(* CODESYS project DBISFactory.project

Project tree, tasks and I/O mapping:
  Device : Berghof MX6 Control, Berghof Automation GmbH, version 1.16.2.0
    application Application
      libraries: Standard, * (System)
      task MainTask (cyclic, interval 4000 µs, priority 0) calls EtherCAT_Master.EtherCAT_Task [EtherCAT_Master.EtherCAT_Task], MAIN
      task EtherCAT_Master (cyclic, interval 4000 µs, priority 0) calls EtherCAT_Master.EtherCAT_Task [EtherCAT_Master.EtherCAT_Task]
      task VISU_TASK (cyclic, interval 100 ms, priority 31) calls VisuElems.Visu_Prg
      global variables SM
      program MAIN [SFC]: FU_Block_active, VG_Block_active, SL_Block_active, TC_active, HR_active, _aInit_active, INIT_BATCH_JOBS_active
      visualisation Visu
      HR/
        global variables HR
        program HR_MULTI_MODE [SFC]: STORE_BOX_active, GET_W_active, WAIT_FOR_VG_TO_PICK_UP_W_active, GET_BOX_active, DECIDE_active, STORE_W_active, WAIT_FOR_VG_TO_BRING_W_active, Init_active, TO_DEFAULT_POS_active
        FBs/
          function block HR_MOVE [ST]
          function block HR_STORE_W [ST]
          function block HR_MOVE_TO_POS [ST]
          function block HR_GET_W [ST]
          function block HR_PUT_W [ST]
          function block HR_TAKE_W [ST]
          function block HR_PUT_W_ON_CONVEYOR [ST]
          function block HR_TAKE_W_FROM_CONVEYOR [ST]
          function block HR_SWITCH_WS [ST]
        program HR_SINGLE_MODE [SFC]: HR_GET_W_active, ConveyorBack_HR_STORE_W_active_exit, HR_STORES_W_active, ConveyorBack_HR_STORE_W_active_active, HR_TO_DEFAULT_POS_active, HR_GET_W_entry, HR_TO_DEFAULT_POS_exit, HR_GETS_W_exit, HR_CONVEYOR_BACKWARD_active, Store_W_active, ToDefaultPos_HR_STORE_W_active_active, HR_WAIT_FOR_TC_active, HR_CONVEYOR_BACKWARD_exit, Init_active, ConveyorBack_HR_STORE_W_active_entry, HR_CALIBRATE_Y_AXIS_active, HR_CALIBRATE_Y_AXIS_exit, HR_CONVEYOR_FORWARD_exit, HR_CONVEYOR_FORWARD_active, HR_STORES_W_exit, HR_SET_TC_STATE_exit, HR_SET_TC_STATE_active
        program HR_SORTING_MODE [SFC]: SORTING_active, TO_DEFAULT_POS_exit, TO_DEFAULT_POS_active, Init_active, HR_SET_TC_STATE_active, HR_SET_TC_STATE_exit, TO_DEFAULT_POS_2_exit, TO_DEFAULT_POS_2_active
      VG/
        FBs/
          function block VG_MOVE [ST]
          function block VG_MOVE_TO_POS [ST]
        program VG_MULTI_MODE [SFC]: TO_DEFAULT_POS_active, DECIDE_active, FROM_HR_TO_FUR_active, TO_SL_TAKE_W_active, TO_HR_PUT_W_active, TO_HR_TAKE_W_active, TO_EJECT_active, Init_active
        program VG_SINGLE_MODE [SFC]: XForward_VG_TAKE_W_active_exit, YUp_VG_DROP_W_active_exit, VG_TO_FU_entry, ZBack_VG_FROM_SL_TO_HR_active_exit, Suction_VG_TAKE_W_active_active, ZBack_VG_TO_FU_active_active, VG_TO_SL_active, YDown_VG_TO_FU_active_exit, ZBack_VG_TO_FU_active_exit_0, Wait_VG_DROP_W_active_active, XForward_VG_TAKE_W_active_active, Wait_VG_TO_FU_active_exit, YDown_VG_DROP_W_active_active, VG_TO_EJECT_POINT_active, YDown_VG_DROP_W_active_exit, OpenVentil_VG_DROP_W_active_exit, VG_EJECT_W_active, OpenVentil_VG_DROP_W_active_active, ZBack_VG_FROM_SL_TO_HR_active_active, ZLeft_AND_XForward_VG_TO_FU_active_active, YDown_VG_TAKE_W_active_exit, YUp_VG_TO_FU_active_exit, YUp_VG_TAKE_W_active_exit, Init_active, YDown_VG_TO_FU_active_active, ZBack_VG_TO_FU_active_exit, YUp_VG_TO_FU_active_active, ZBack_VG_TAKE_W_active_exit, VG_TO_FU_active, OpenVentil_VG_TO_FU_active_active, YUp_VG_DROP_W_active_active, ZBack_VG_TAKE_W_active_active, VG_TAKE_W_entry, Wait_VG_TO_FU_active_active, YUp_VG_TAKE_W_active_active, VG_DROP_W_entry, VG_TO_DEFAULT_POS_active, VG_DROP_W_active, VG_TAKE_W_active, YDown_VG_TAKE_W_active_active, Wait_VG_DROP_W_active_exit, VG_DROP_W_exit, VG_FROM_SL_TO_HR_active, VG_TO_HR_active, ZBack_VG_TO_FU_active_active_0, ZLeft_AND_XForward_VG_TO_FU_active_exit, VG_WAIT_FOR_SL_active, VG_WAIT_FOR_SL_exit, VG_YUp_active, VG_YUp_exit, VG_TO_EJECT_POINT_exit, VG_EJECT_active, VG_EJECT_exit, BACK_TO_DEFAULT_active, VG_TO_SL_exit, VG_DIRECTLY_EJECT_W_active, VG_TO_HR_exit
        global variables VG
      FUR/
        program FUR_SINGLE_MODE [SFC]: FUR_SUCCER_UP_active_0, FUR_SUCCER_TO_ROTATION_DESK_active, FUR_SAW_active, FUR_WAIT_FOR_W_exit, Init_active, FUR_SUCCER_DOWN2_active, FUR_SUCCER_DOWN_active, FUR_TO_CONVEYOR_active, FUR_SUCCER_UP_active, FUR_TO_DEFAULT_POS_active, FUR_WAIT_FOR_W_active, FUR_BURN_active
        program FUR_MULTI_MODE [SFC]: BURNER_active, SUCCER_active, SAW_active, TO_DEFAULT_POS_active, TO_DEFAULT_POS_exit
        global variables FUR
        FBs/
          function block FUR_BURN [ST]
      SL/
        program SL_SINGLE_MODE [SFC]: Init_active, SL_GO_active
        global variables SL
        program SL_MULTI_MODE [SFC]: SL_GO_active, Init_active
        FBs/
          function block SL_FB [SFC]: Init_active, SL_COLORCHECK_active, SL_GET_VALUE_active, SL_PASS_LBEntry_active, SL_PASS_LBEntry_exit, SL_PULS_COUNTER_active, SL_PULS_COUNTER_exit, SL_SORTING_active, SL_STOREROOM_active
      TC/
        FUNs/
          function addBatchJobToQueue [ST]
          function newWorkpiece [ST]
          function addWorkpieceToBatchJob [ST]
          function newFormat [ST]
          function newBatchJob [ST]
        global variables TC
        program TC_POU [SFC]: Decide_next_W_or_BatchJob_active, Set_Workpiece_active, start_batch_job_active, Init_active, Next_W_active, Next_W_exit, Decide_next_W_or_BatchJob_exit, Start_Batch_Job_exit
      datastructures/
        Enums/
          data type ExecutionMode
          data type RackPos
          States/
            data type BatchJobState
            data type HR_State
            data type VG_State
            data type FUR_State
            data type SL_State
            data type W_State
            data type TC_State
        Structs/
          data type Format
          data type BatchJobQueue
          data type Workpiece
          data type BatchJob
      Symbols
    Extension_Slots : Extension Slots, Berghof Automation GmbH, order no. 
      , version 1.0.0.0
      <Leer>
      Berghof_IO : Berghof IO, Berghof Automation GmbH, order no. 
      , version 1.1.0.0
          unmapped channels: Digital Input 0, Digital Input 1, Digital Input 2, Digital Input 3, Digital Input 4, Digital Output 0, Digital Output 1, Digital Output 2, Digital Output 3, Digital Output 4, Channel 0, Channel 1, Channel 2, Channel 3, Channel 4, Channel 5, Channel 6, Channel 7, Channel 8, Channel 9, Channel 10, Channel 11, Channel 0, Channel 1, Channel 2, Channel 3, Channel 4, Channel 5, Channel 6, Channel 7, Counter/Encoder 0, Counter/Encoder 1, Counter/Encoder 2, DUMMY 0
    EtherCAT_Master : EtherCAT Master, 3S - Smart Software Solutions GmbH, version 3.5.10.0
        settings: SlaveAutoRestart = True; NetworkName = 'eth1'; SelectNetworkByName = True
      ECC_DIO_16_16P : ECC DIO 16/16 P (250 000 600), Berghof Automation GmbH, version Revision=16#00000001
          settings: DC sync0 cycletime = 4000; DC sync1 cycletime = 4000
          unmapped channels: Digital Output 0, Digital Output 1, Digital Input 0, Digital Input 1
  libraries: VisuSymbols, 3.5.10.0 (System)
  text list GlobalTextList
*)

// Device/Application/datastructures/Enums/States/BatchJobState
(*
	States of a BatchJob

Copyright (c) 2019 Manuel Goester, Michael Witt, Klaus Kammerer
Institute of Databases and Information Systems, Ulm University, Germany

Permission is hereby granted, free of charge, to any person obtaining a copy 
of this software and associated documentation files (the "Software"), to deal 
in the Software without restriction, including without limitation the rights 
to use, copy, modify, merge, publish, distribute, sublicense, and/or sell 
copies of the Software, and to permit persons to whom the Software is 
furnished to do so, subject to the following conditions:

The above copyright notice and this permission notice shall be included in 
all copies or substantial portions of the Software.

THE SOFTWARE IS PROVIDED "AS IS", WITHOUT WARRANTY OF ANY KIND, EXPRESS OR 
IMPLIED, INCLUDING BUT NOT LIMITED TO THE WARRANTIES OF MERCHANTABILITY, 
FITNESS FOR A PARTICULAR PURPOSE AND NONINFRINGEMENT. IN NO EVENT SHALL THE 
AUTHORS OR COPYRIGHT HOLDERS BE LIABLE FOR ANY CLAIM, DAMAGES OR OTHER 
LIABILITY, WHETHER IN AN ACTION OF CONTRACT, TORT OR OTHERWISE, ARISING FROM, 
OUT OF OR IN CONNECTION WITH THE SOFTWARE OR THE USE OR OTHER DEALINGS 
IN THE SOFTWARE.
*)
TYPE BatchJobState :
(
	// NULL always expresses that the object has not been initialized yet
	NULL := 0,
	
	// BatchJob has been initialized and is waiting to be executed
	WAITING := 1,
	
	// BatchJob has been started and is being executed now
	STARTED := 2,
	
	// BatchJob has been paused during execution
	PAUSED := 3,
	
	// BatchJob has been aborted. This may happen at any time
	ABORTED := 4,
	
	// BatchJob has been finished
	FINISHED := 5
);
END_TYPE

// Device/Application/datastructures/Enums/ExecutionMode
(*
	Execution modes of a BatchJob
	
Copyright (c) 2019 Manuel Goester, Michael Witt, Klaus Kammerer
Institute of Databases and Information Systems, Ulm University, Germany

Permission is hereby granted, free of charge, to any person obtaining a copy 
of this software and associated documentation files (the "Software"), to deal 
in the Software without restriction, including without limitation the rights 
to use, copy, modify, merge, publish, distribute, sublicense, and/or sell 
copies of the Software, and to permit persons to whom the Software is 
furnished to do so, subject to the following conditions:

The above copyright notice and this permission notice shall be included in 
all copies or substantial portions of the Software.

THE SOFTWARE IS PROVIDED "AS IS", WITHOUT WARRANTY OF ANY KIND, EXPRESS OR 
IMPLIED, INCLUDING BUT NOT LIMITED TO THE WARRANTIES OF MERCHANTABILITY, 
FITNESS FOR A PARTICULAR PURPOSE AND NONINFRINGEMENT. IN NO EVENT SHALL THE 
AUTHORS OR COPYRIGHT HOLDERS BE LIABLE FOR ANY CLAIM, DAMAGES OR OTHER 
LIABILITY, WHETHER IN AN ACTION OF CONTRACT, TORT OR OTHERWISE, ARISING FROM, 
OUT OF OR IN CONNECTION WITH THE SOFTWARE OR THE USE OR OTHER DEALINGS 
IN THE SOFTWARE.
*)
TYPE ExecutionMode :
(
	single := 0,
	multi := 1,
	sorting := 2
);
END_TYPE

// Device/Application/datastructures/Structs/Format
(*
	A Format defines the execution options of a workpiece

Copyright (c) 2019 Manuel Goester, Michael Witt, Klaus Kammerer
Institute of Databases and Information Systems, Ulm University, Germany

Permission is hereby granted, free of charge, to any person obtaining a copy 
of this software and associated documentation files (the "Software"), to deal 
in the Software without restriction, including without limitation the rights 
to use, copy, modify, merge, publish, distribute, sublicense, and/or sell 
copies of the Software, and to permit persons to whom the Software is 
furnished to do so, subject to the following conditions:

The above copyright notice and this permission notice shall be included in 
all copies or substantial portions of the Software.

THE SOFTWARE IS PROVIDED "AS IS", WITHOUT WARRANTY OF ANY KIND, EXPRESS OR 
IMPLIED, INCLUDING BUT NOT LIMITED TO THE WARRANTIES OF MERCHANTABILITY, 
FITNESS FOR A PARTICULAR PURPOSE AND NONINFRINGEMENT. IN NO EVENT SHALL THE 
AUTHORS OR COPYRIGHT HOLDERS BE LIABLE FOR ANY CLAIM, DAMAGES OR OTHER 
LIABILITY, WHETHER IN AN ACTION OF CONTRACT, TORT OR OTHERWISE, ARISING FROM, 
OUT OF OR IN CONNECTION WITH THE SOFTWARE OR THE USE OR OTHER DEALINGS 
IN THE SOFTWARE.
*)
TYPE Format :
STRUCT
	furEnabled: BOOL;
	sawEnabled: BOOL;
	colorCheckEnabled: BOOL;
	ejectEnabled: BOOL;
	
	furDuration: TIME;
	sawDuration: TIME;
END_STRUCT
END_TYPE

// Device/Application/datastructures/Structs/BatchJobQueue
(*
	Configured BatchJobs are stored in a BatchJobQueue

Copyright (c) 2019 Manuel Goester, Michael Witt, Klaus Kammerer
Institute of Databases and Information Systems, Ulm University, Germany

Permission is hereby granted, free of charge, to any person obtaining a copy 
of this software and associated documentation files (the "Software"), to deal 
in the Software without restriction, including without limitation the rights 
to use, copy, modify, merge, publish, distribute, sublicense, and/or sell 
copies of the Software, and to permit persons to whom the Software is 
furnished to do so, subject to the following conditions:

The above copyright notice and this permission notice shall be included in 
all copies or substantial portions of the Software.

THE SOFTWARE IS PROVIDED "AS IS", WITHOUT WARRANTY OF ANY KIND, EXPRESS OR 
IMPLIED, INCLUDING BUT NOT LIMITED TO THE WARRANTIES OF MERCHANTABILITY, 
FITNESS FOR A PARTICULAR PURPOSE AND NONINFRINGEMENT. IN NO EVENT SHALL THE 
AUTHORS OR COPYRIGHT HOLDERS BE LIABLE FOR ANY CLAIM, DAMAGES OR OTHER 
LIABILITY, WHETHER IN AN ACTION OF CONTRACT, TORT OR OTHERWISE, ARISING FROM, 
OUT OF OR IN CONNECTION WITH THE SOFTWARE OR THE USE OR OTHER DEALINGS 
IN THE SOFTWARE.
*)
TYPE BatchJobQueue :
STRUCT
	// batch job queue
	batchJobs: ARRAY [1..512] OF BatchJob;
	
	// next free place in batchJobs
	nextFreePos: INT := 1;
	
	// amount of batch jobs currently being in queue
	amountBatchJobs: INT := 0;
	
	// true if batchJobs array full
	full: BOOL;
END_STRUCT
END_TYPE

// Device/Application/datastructures/Structs/Workpiece
(*
	Datastructure describing the "real world workpiece"

Copyright (c) 2019 Manuel Goester, Michael Witt, Klaus Kammerer
Institute of Databases and Information Systems, Ulm University, Germany

Permission is hereby granted, free of charge, to any person obtaining a copy 
of this software and associated documentation files (the "Software"), to deal 
in the Software without restriction, including without limitation the rights 
to use, copy, modify, merge, publish, distribute, sublicense, and/or sell 
copies of the Software, and to permit persons to whom the Software is 
furnished to do so, subject to the following conditions:

The above copyright notice and this permission notice shall be included in 
all copies or substantial portions of the Software.

THE SOFTWARE IS PROVIDED "AS IS", WITHOUT WARRANTY OF ANY KIND, EXPRESS OR 
IMPLIED, INCLUDING BUT NOT LIMITED TO THE WARRANTIES OF MERCHANTABILITY, 
FITNESS FOR A PARTICULAR PURPOSE AND NONINFRINGEMENT. IN NO EVENT SHALL THE 
AUTHORS OR COPYRIGHT HOLDERS BE LIABLE FOR ANY CLAIM, DAMAGES OR OTHER 
LIABILITY, WHETHER IN AN ACTION OF CONTRACT, TORT OR OTHERWISE, ARISING FROM, 
OUT OF OR IN CONNECTION WITH THE SOFTWARE OR THE USE OR OTHER DEALINGS 
IN THE SOFTWARE.
*)
TYPE Workpiece :
STRUCT
	// red, blue, white or unknown
	color: STRING[7];
	
	// 0 = high rack, 1 = vacuum gripper, 2 = Furnace, 3 = sorting line
	linePos: INT;
	
	// position in high rack at begin and end of batch job
	// (1,1) (1,2) (1,3)
	// (2,1) (2,2) (2,3)
	// (3,1) (3,2) (3,3)
	//highRackPos: ARRAY [1..2] OF INT;
	//highRackPosEnd: ARRAY [1..2] OF INT;
	
	// position in sorting line
	sortingLinePos: INT;
	
	state: W_State;	
	startPos: RackPos;
	endPos: RackPos;
	
	// defines which actions will be executed and how long
	format: Format;
END_STRUCT
END_TYPE

// Device/Application/datastructures/Structs/BatchJob
(*
	A BatchJob is a task which shall be executed on the production lane. 
	It consists of a set of workpieces, which are executed by the production lane in a certain mode.

Copyright (c) 2019 Manuel Goester, Michael Witt, Klaus Kammerer
Institute of Databases and Information Systems, Ulm University, Germany

Permission is hereby granted, free of charge, to any person obtaining a copy 
of this software and associated documentation files (the "Software"), to deal 
in the Software without restriction, including without limitation the rights 
to use, copy, modify, merge, publish, distribute, sublicense, and/or sell 
copies of the Software, and to permit persons to whom the Software is 
furnished to do so, subject to the following conditions:

The above copyright notice and this permission notice shall be included in 
all copies or substantial portions of the Software.

THE SOFTWARE IS PROVIDED "AS IS", WITHOUT WARRANTY OF ANY KIND, EXPRESS OR 
IMPLIED, INCLUDING BUT NOT LIMITED TO THE WARRANTIES OF MERCHANTABILITY, 
FITNESS FOR A PARTICULAR PURPOSE AND NONINFRINGEMENT. IN NO EVENT SHALL THE 
AUTHORS OR COPYRIGHT HOLDERS BE LIABLE FOR ANY CLAIM, DAMAGES OR OTHER 
LIABILITY, WHETHER IN AN ACTION OF CONTRACT, TORT OR OTHERWISE, ARISING FROM, 
OUT OF OR IN CONNECTION WITH THE SOFTWARE OR THE USE OR OTHER DEALINGS 
IN THE SOFTWARE.
*)
TYPE BatchJob :
STRUCT
	// amount of workpieces in batch job
	batchSize: INT;
	
	// workpieces being processed
	workpieces: ARRAY [1..9] OF Workpiece;
	
	// next free place in workpieces
	nextFreeWPos: INT := 1;
	
	// index in workpieces of the next workpiece whose production has not started yet
	nextNotProcessedIdx: INT := 1;
	
	// states how many workpieces are already finished
	amountFinishedW: INT := 0;
	
	// type of execution
	mode: ExecutionMode := ExecutionMode.single;
	
	// time when created
	timeCreated: DATE_AND_TIME;
	
	// time when started
	timeStarted: DATE_AND_TIME;
	
	// time when finished / aborted
	timeFinished: DATE_AND_TIME;
	
	// states the time how long the batch job was in pause state
	pauseDuration: TIME;
	
	// states how long the batch job took 
	duration: TIME;
	
	// state of batch job
	state: BatchJobState := BatchJobState.NULL;
END_STRUCT
END_TYPE

// Device/Application/datastructures/Enums/RackPos
(*
	Positions in high rack. Used for HR navigation

Copyright (c) 2019 Manuel Goester, Michael Witt, Klaus Kammerer
Institute of Databases and Information Systems, Ulm University, Germany

Permission is hereby granted, free of charge, to any person obtaining a copy 
of this software and associated documentation files (the "Software"), to deal 
in the Software without restriction, including without limitation the rights 
to use, copy, modify, merge, publish, distribute, sublicense, and/or sell 
copies of the Software, and to permit persons to whom the Software is 
furnished to do so, subject to the following conditions:

The above copyright notice and this permission notice shall be included in 
all copies or substantial portions of the Software.

THE SOFTWARE IS PROVIDED "AS IS", WITHOUT WARRANTY OF ANY KIND, EXPRESS OR 
IMPLIED, INCLUDING BUT NOT LIMITED TO THE WARRANTIES OF MERCHANTABILITY, 
FITNESS FOR A PARTICULAR PURPOSE AND NONINFRINGEMENT. IN NO EVENT SHALL THE 
AUTHORS OR COPYRIGHT HOLDERS BE LIABLE FOR ANY CLAIM, DAMAGES OR OTHER 
LIABILITY, WHETHER IN AN ACTION OF CONTRACT, TORT OR OTHERWISE, ARISING FROM, 
OUT OF OR IN CONNECTION WITH THE SOFTWARE OR THE USE OR OTHER DEALINGS 
IN THE SOFTWARE.
*)
TYPE RackPos :
(
	NULL := 0,
	RACK_11 := 1,
	RACK_12 := 2,
	RACK_13 := 3,
	RACK_21 := 4,
	RACK_22 := 5,
	RACK_23 := 6,
	RACK_31 := 7,
	RACK_32 := 8,
	RACK_33 := 9,
	
	CONVEYOR := 10,
	
	// there are different values for up position or down position at rack or at conveyor
	// see: HR_FBs/HR_MOVE_TO_POS
	UP := 11,
	DOWN := 12	
);
END_TYPE

// Device/Application/datastructures/Enums/States/HR_State
(*
	States of the HR (High Rack) station.

Copyright (c) 2019 Manuel Goester, Michael Witt, Klaus Kammerer
Institute of Databases and Information Systems, Ulm University, Germany

Permission is hereby granted, free of charge, to any person obtaining a copy 
of this software and associated documentation files (the "Software"), to deal 
in the Software without restriction, including without limitation the rights 
to use, copy, modify, merge, publish, distribute, sublicense, and/or sell 
copies of the Software, and to permit persons to whom the Software is 
furnished to do so, subject to the following conditions:

The above copyright notice and this permission notice shall be included in 
all copies or substantial portions of the Software.

THE SOFTWARE IS PROVIDED "AS IS", WITHOUT WARRANTY OF ANY KIND, EXPRESS OR 
IMPLIED, INCLUDING BUT NOT LIMITED TO THE WARRANTIES OF MERCHANTABILITY, 
FITNESS FOR A PARTICULAR PURPOSE AND NONINFRINGEMENT. IN NO EVENT SHALL THE 
AUTHORS OR COPYRIGHT HOLDERS BE LIABLE FOR ANY CLAIM, DAMAGES OR OTHER 
LIABILITY, WHETHER IN AN ACTION OF CONTRACT, TORT OR OTHERWISE, ARISING FROM, 
OUT OF OR IN CONNECTION WITH THE SOFTWARE OR THE USE OR OTHER DEALINGS 
IN THE SOFTWARE.
*)
TYPE HR_State :
(
	// NULL always expresses that the Object has not been initialized yet
	NULL := 0,
	
	// used in single mode
	AT_DEFAULT_POS := 1,
	FINISHED_SINGLE_MODE := 2,
	AT_CONVEYOR_BOX_FULL := 25,
	AT_CONVEYOR_BOX_EMPTY := 26,
	
	// used in multi mode
	WAIT_FOR_VG_TO_BRING_W := 8,
	GET_W := 9, // <-- also used in single mode
	GET_BOX := 10,
	STORE_W := 20,
	STORE_BOX := 19,
	WAIT_FOR_VG_TO_PICK_UP_W := 11,
	READY := 12,
	
	// used in sorting mode
	FINISHED_SORTING_MODE := 40,
	SORTING := 41
);
END_TYPE

// Device/Application/datastructures/Enums/States/VG_State
(*
	States of the VG (Vacuum Gripper) station.

Copyright (c) 2019 Manuel Goester, Michael Witt, Klaus Kammerer
Institute of Databases and Information Systems, Ulm University, Germany

Permission is hereby granted, free of charge, to any person obtaining a copy 
of this software and associated documentation files (the "Software"), to deal 
in the Software without restriction, including without limitation the rights 
to use, copy, modify, merge, publish, distribute, sublicense, and/or sell 
copies of the Software, and to permit persons to whom the Software is 
furnished to do so, subject to the following conditions:

The above copyright notice and this permission notice shall be included in 
all copies or substantial portions of the Software.

THE SOFTWARE IS PROVIDED "AS IS", WITHOUT WARRANTY OF ANY KIND, EXPRESS OR 
IMPLIED, INCLUDING BUT NOT LIMITED TO THE WARRANTIES OF MERCHANTABILITY, 
FITNESS FOR A PARTICULAR PURPOSE AND NONINFRINGEMENT. IN NO EVENT SHALL THE 
AUTHORS OR COPYRIGHT HOLDERS BE LIABLE FOR ANY CLAIM, DAMAGES OR OTHER 
LIABILITY, WHETHER IN AN ACTION OF CONTRACT, TORT OR OTHERWISE, ARISING FROM, 
OUT OF OR IN CONNECTION WITH THE SOFTWARE OR THE USE OR OTHER DEALINGS 
IN THE SOFTWARE.
*)
TYPE VG_State :
(
	// NULL always expresses that the object has not been initialized yet
	NULL := 0,
	
	// used in single mode
	FROM_HR_TO_EJECT := 6,
	AT_HR := 30,
	FROM_HR_TO_FUR := 31,
	AT_SL_OUTPUT_1 := 32,
	AT_SL_OUTPUT_2 := 33,
	AT_SL_OUTPUT_3 := 34,
	WAIT_FOR_SL := 35,
	AT_EJECT_1 := 36,
	AT_EJECT_2 := 37,
	AT_EJECT_3 := 38,
	TO_SL_OUTPUT_1 := 39,
	TO_SL_OUTPUT_2 := 40,
	TO_SL_OUTPUT_3 := 41,
	FROM_DEFAULT_POS_TO_HR := 43,
	GET_W_FROM_HR := 44,
	ABOVE_SL := 56,
	FROM_SL_TO_HR := 57,
	DROPPING_W_TO_HR := 59,
	
	// used in multi mode
	TO_FUR_PUT_W := 8,
	TO_FUR_PUT_W_FINISHED := 9,
	TO_SL_TAKE_W := 10,
	TO_SL_TAKE_W_FINISHED := 11,
	TO_HR_PUT_W := 12,
	TO_HR_PUT_W_FINISHED := 13,
	TO_HR_TAKE_W := 14,
	TO_HR_TAKE_W_FINISHED := 15,
	TO_EJECT := 16,
	TO_EJECT_FINISHED := 17,
	TO_SL := 45,
	// ready if VG is at default pos or if VG put down a workpiece at HR --> VG is ready for next workpiece
	READY := 18,
	
	// used in single and multi mode
	AT_DEFAULT_POS := 1,
	TO_DEFAULT_POS := 5
);
END_TYPE

// Device/Application/datastructures/Enums/States/FUR_State
(*
	States of the FUR (Furnace) station.
	The station is composed of a burner, succer, rotary desk and saw.

Copyright (c) 2019 Manuel Goester, Michael Witt, Klaus Kammerer
Institute of Databases and Information Systems, Ulm University, Germany

Permission is hereby granted, free of charge, to any person obtaining a copy 
of this software and associated documentation files (the "Software"), to deal 
in the Software without restriction, including without limitation the rights 
to use, copy, modify, merge, publish, distribute, sublicense, and/or sell 
copies of the Software, and to permit persons to whom the Software is 
furnished to do so, subject to the following conditions:

The above copyright notice and this permission notice shall be included in 
all copies or substantial portions of the Software.

THE SOFTWARE IS PROVIDED "AS IS", WITHOUT WARRANTY OF ANY KIND, EXPRESS OR 
IMPLIED, INCLUDING BUT NOT LIMITED TO THE WARRANTIES OF MERCHANTABILITY, 
FITNESS FOR A PARTICULAR PURPOSE AND NONINFRINGEMENT. IN NO EVENT SHALL THE 
AUTHORS OR COPYRIGHT HOLDERS BE LIABLE FOR ANY CLAIM, DAMAGES OR OTHER 
LIABILITY, WHETHER IN AN ACTION OF CONTRACT, TORT OR OTHERWISE, ARISING FROM, 
OUT OF OR IN CONNECTION WITH THE SOFTWARE OR THE USE OR OTHER DEALINGS 
IN THE SOFTWARE.
*)
TYPE FUR_State :
(
	// TODO : Use these states also in multi mode
	
	// NULL always expresses that the Object has not been initialized yet
	NULL := 0,
	
	// used in single mode
	// FUR is ready to take a new workpiece
	FUR_WAITING_FOR_W := 1,	
	// Workpiece passed the lightbarrier at waggon
	FUR_LB_PASSED := 2,
	
	// used in single and multi mode
	// Wagon is inside of burner
	FUR_WAGON_INSIDE := 3,
	// Furnace is finished with buring the workpiece
	FUR_BURNED := 4,
	// Wagon is outside of burner
	FUR_WAGON_OUTSIDE := 5,	
	
	// used in single mode
	// furnace succer is at furnace
	FUR_SUCCER_AT_FUR := 6,
	// furnace succer picks up workpiece
	FUR_SUCCER_DOWN_AT_FUR := 7,
	FUR_SUCCER_UP_AT_FUR := 8,
	// furnace succer on the way to rotary desk
	FUR_SUCCER_TO_ROTARY_DESK := 9,
	// furnace succer at rotary desk
	FUR_SUCCER_AT_ROTARY_DESK := 10,
	// furnace succer puts down workpiece
	FUR_SUCCER_DOWN_AT_RD := 11,
	FUR_SUCCER_UP_AT_RD := 12,
	// saw has been finished
	FUR_SAW_FINISHED := 13,	
	// saw has been skipped			
	FUR_SKIP_SAW := 14,
	// station has finished processing this workpiece
	FUR_W_FINISHED_BACK_TO_DEFAULT := 15
);
END_TYPE

// Device/Application/datastructures/Enums/States/SL_State
(*
	States of the SL (Sorting Line) station.

Copyright (c) 2019 Manuel Goester, Michael Witt, Klaus Kammerer
Institute of Databases and Information Systems, Ulm University, Germany

Permission is hereby granted, free of charge, to any person obtaining a copy 
of this software and associated documentation files (the "Software"), to deal 
in the Software without restriction, including without limitation the rights 
to use, copy, modify, merge, publish, distribute, sublicense, and/or sell 
copies of the Software, and to permit persons to whom the Software is 
furnished to do so, subject to the following conditions:

The above copyright notice and this permission notice shall be included in 
all copies or substantial portions of the Software.

THE SOFTWARE IS PROVIDED "AS IS", WITHOUT WARRANTY OF ANY KIND, EXPRESS OR 
IMPLIED, INCLUDING BUT NOT LIMITED TO THE WARRANTIES OF MERCHANTABILITY, 
FITNESS FOR A PARTICULAR PURPOSE AND NONINFRINGEMENT. IN NO EVENT SHALL THE 
AUTHORS OR COPYRIGHT HOLDERS BE LIABLE FOR ANY CLAIM, DAMAGES OR OTHER 
LIABILITY, WHETHER IN AN ACTION OF CONTRACT, TORT OR OTHERWISE, ARISING FROM, 
OUT OF OR IN CONNECTION WITH THE SOFTWARE OR THE USE OR OTHER DEALINGS 
IN THE SOFTWARE.
*)
TYPE SL_State :
(
	
	// NULL always expresses that the object has not been initialized yet
	NULL := 0,
	
	// SL is ready to process a new workpiece
	WAITING_FOR_W := 1,
	// Lightbarrier at SL entry has been passed by a workpiece
	W_AT_LB := 2,

	W_AT_COLORCHECK := 3,
	COLORCHECK_FINISHED := 4,
	W_READY_FOR_SORTING := 5,
	// if no color was detected, the workpiece will be thrown out to trash 
	THROW_OUT := 6,
	
	SORTING := 7,
	WAITING_FOR_VG_TO_PICK_UP_W	 := 8,
	EJECT := 9,
	EJECTED := 10,
	
	// SL got a workpiece to process it
	W_RECEIVED := 11
);
END_TYPE

// Device/Application/datastructures/Enums/States/W_State
(*
	Workpiece States

Copyright (c) 2019 Manuel Goester, Michael Witt, Klaus Kammerer
Institute of Databases and Information Systems, Ulm University, Germany

Permission is hereby granted, free of charge, to any person obtaining a copy 
of this software and associated documentation files (the "Software"), to deal 
in the Software without restriction, including without limitation the rights 
to use, copy, modify, merge, publish, distribute, sublicense, and/or sell 
copies of the Software, and to permit persons to whom the Software is 
furnished to do so, subject to the following conditions:

The above copyright notice and this permission notice shall be included in 
all copies or substantial portions of the Software.

THE SOFTWARE IS PROVIDED "AS IS", WITHOUT WARRANTY OF ANY KIND, EXPRESS OR 
IMPLIED, INCLUDING BUT NOT LIMITED TO THE WARRANTIES OF MERCHANTABILITY, 
FITNESS FOR A PARTICULAR PURPOSE AND NONINFRINGEMENT. IN NO EVENT SHALL THE 
AUTHORS OR COPYRIGHT HOLDERS BE LIABLE FOR ANY CLAIM, DAMAGES OR OTHER 
LIABILITY, WHETHER IN AN ACTION OF CONTRACT, TORT OR OTHERWISE, ARISING FROM, 
OUT OF OR IN CONNECTION WITH THE SOFTWARE OR THE USE OR OTHER DEALINGS 
IN THE SOFTWARE.
*)
TYPE W_State :
(
	// NULL always expresses that the object has not been initialized yet
	NULL := 0,
	
	// states at HR
	AT_RACK_11 := 111,
	AT_RACK_12 := 112,
	AT_RACK_13 := 113,
	AT_RACK_21 := 121,
	AT_RACK_22 := 122,
	AT_RACK_23 := 123,
	AT_RACK_31 := 131,
	AT_RACK_32 := 132,
	AT_RACK_33 := 133,
	
	// NOT used
	FROM_RACK_TO_CONVEYOR := 140,
	AT_CONVEYOR_INSIDE := 141,
	FROM_CONVEYOR_INSIDE_TO_OUTSIDE := 142,
	AT_CONVEYOR_OUTSIDE := 143,
	FROM_CONVEYOR_OUTSIDE_TO_INSIDE := 144,
	
	// states at VG
	// NOT used
	AT_HR := 200,
	FROM_HR_TO_FUR := 201,
	FROM_SL_OUTPUT_TO_HR := 202,
	FROM_SL_OUTPUT_1_TO_HR := 203,
	FROM_SL_OUTPUT_2_TO_HR := 204,
	FROM_SL_OUTPUT_3_TO_HR := 205,
	FROM_SL_TO_EJECT := 206,
	FROM_SL_OUTPUT_1_TO_EJECT := 207,
	FROM_SL_OUTPUT_2_TO_EJECT := 208,
	FROM_SL_OUTPUT_3_TO_EJECT := 209,
	FROM_FUR_TO_HR := 210,
	
	// states at FUR
	AT_FUR_IN_WAGON := 300,
	AT_FUR_IN_FUR := 301,
	AT_FUR_ATTACHED_TO_SUCCER := 302,
	AT_FUR_ON_ROTARY_DESK := 303,
	AT_FUR_AT_SAW := 304,
	AT_FUR_ON_CONVEYOR := 305,
	
	// states at SL
	// not used
	AT_SL_AT_ENTRY_LIGHT_BARRIER := 400,
	AT_SL_AT_COLORCHECK := 401,
	AT_SL_AT_EXIT_LIGHT_BARRIER := 402,
	AT_SL_OUTPUT_1 := 403,
	AT_SL_OUTPUT_2 := 404,
	AT_SL_OUTPUT_3 := 405,
	AT_SL_OUTPUT_TRASH := 406,
	
	// states at EJECT point
	// not used
	AT_EJECT_1 := 500,
	AT_EJECT_2 := 501,
	AT_EJECT_3 := 502
);
END_TYPE

// Device/Application/datastructures/Enums/States/TC_State
(*
	States of TC (Task Configurator).

Copyright (c) 2019 Manuel Goester, Michael Witt, Klaus Kammerer
Institute of Databases and Information Systems, Ulm University, Germany

Permission is hereby granted, free of charge, to any person obtaining a copy 
of this software and associated documentation files (the "Software"), to deal 
in the Software without restriction, including without limitation the rights 
to use, copy, modify, merge, publish, distribute, sublicense, and/or sell 
copies of the Software, and to permit persons to whom the Software is 
furnished to do so, subject to the following conditions:

The above copyright notice and this permission notice shall be included in 
all copies or substantial portions of the Software.

THE SOFTWARE IS PROVIDED "AS IS", WITHOUT WARRANTY OF ANY KIND, EXPRESS OR 
IMPLIED, INCLUDING BUT NOT LIMITED TO THE WARRANTIES OF MERCHANTABILITY, 
FITNESS FOR A PARTICULAR PURPOSE AND NONINFRINGEMENT. IN NO EVENT SHALL THE 
AUTHORS OR COPYRIGHT HOLDERS BE LIABLE FOR ANY CLAIM, DAMAGES OR OTHER 
LIABILITY, WHETHER IN AN ACTION OF CONTRACT, TORT OR OTHERWISE, ARISING FROM, 
OUT OF OR IN CONNECTION WITH THE SOFTWARE OR THE USE OR OTHER DEALINGS 
IN THE SOFTWARE.
*)
TYPE TC_State :
(
	// NULL always expresses that the Object has not been initialized yet
	NULL := 0,
	
	// TC has loaded a new workpiece to HR
	W_LOADED := 1,
	// TC is waiting until the workpiece has been processed
	WAIT_UNTIL_W_FINISHED := 2,
	
	// TC is loading a new workpiece
	LOAD_NEXT_W := 3
);
END_TYPE

// Device/Application/TC/TC
VAR_GLOBAL
	// the mode thats currently active
	mode_active: ExecutionMode;
	
	// true if program started
	is_plc_running: BOOL;
	
	// true if user has selected
	instant_shutdown AT %IX1.7: BOOL;
	
	// global batch job queue 
	batchJobQueue: BatchJobQueue;
	
	// the index in batchJobs of the batch job which is currently running
	currBatchJobIdx: INT := 1;
	
	// state of Task configuration
	state: TC_State;
	
	// This is a workpiece being used as an NULL object in Java
	nullW: Workpiece;
	
	// This is a BatchJob being used as an NULL object in Java
	nullB: BatchJob;
END_VAR

// Device/Application/SM
VAR_GLOBAL
	// SM = single mode
	// current workpiece being processed in single mode
	currW: Workpiece;
END_VAR

// Device/Application/HR/HR
VAR_GLOBAL
	//------------------------------------------------------------------------------------//
	//--------------------------------------INPUTS----------------------------------------//
	//------------------------------------------------------------------------------------//
	sHorizontal AT %IX0.0: BOOL;
	lbIn AT %IX0.1: BOOL;
	lbOut AT %IX0.2: BOOL;
	sVertical AT %IX0.3: BOOL;
	sCFront AT %IX0.4: BOOL;
	sCBack AT %IX0.5: BOOL;
	encHorizontal AT %IX1.1: BOOL;
	encVertical AT %IX1.2: BOOL;
	
	//------------------------------------------------------------------------------------//
	//--------------------------------------OUTPUTS---------------------------------------//
	//------------------------------------------------------------------------------------//
	mCbForward AT %QX0.0: BOOL;
	mCbBackward AT %QX0.1: BOOL;
	mHorizontalLeft AT %QX0.2: BOOL;
	mHorizontalRight AT %QX0.3: BOOL;
	mVerticalDown AT %QX0.4: BOOL;
	mVerticalUp AT %QX0.5: BOOL;
	mCForward AT %QX0.6: BOOL;
	mCBackward AT %QX0.7: BOOL;
	
	//------------------------------------------------------------------------------------//
	//------------------------------------PROGRAM VARS------------------------------------//
	//------------------------------------------------------------------------------------//
	// the state in which HR currently is
	state: HR_State;
	
	// true if the start button at Visu is pressed
	started_btn_is_pressed: BOOL;
	
	// true if any motor of HR is running
	any_motor_running: BOOL;
	
	// flag needed for decision making in multi mode
	decidedToTakeANewW: BOOL;
	
	// these counters define the current position of HR
	cX: INT;
	cY: INT;
	
	// current BatchJob and workpiece index being processed at HR
	bIdx: INT;
	wIdx: INT;
	currW: Workpiece;
END_VAR

// Device/Application/FUR/FUR
VAR_GLOBAL
	//------------------------------------------------------------------------------------//
	//--------------------------------------INPUTS----------------------------------------//
	//------------------------------------------------------------------------------------//
	sRaPosSucker AT %IX300.0: BOOL;
	sRaPosConveyorBelt AT %IX300.1: BOOL;
	lbConveyorBelt AT %IX300.2: BOOL;
	sRaPosSaw AT %IX300.3: BOOL;
	sSuckerPosRa AT %IX300.4: BOOL;
	sFurnanceSliderInside AT %IX300.5: BOOL;
	sFurnanceSliderOutside AT %IX300.6: BOOL;
	sSuckerPosFF AT %IX300.7: BOOL;
	lbFurnance AT %IX301.0: BOOL;
	
	//------------------------------------------------------------------------------------//
	//--------------------------------------OUTPUTS---------------------------------------//
	//------------------------------------------------------------------------------------//	
	mRaClockwise AT %QX40.0: BOOL;
	mRaCClockwise AT %QX40.1: BOOL;
	mConveyorBeltForward AT %QX40.2: BOOL;
	mSaw AT %QX40.3: BOOL;
	mFurnanceSliderIn AT %QX40.4: BOOL;
	mFurnanceSliderOut AT %QX40.5: BOOL;
	mSuckertoFurnance AT %QX40.6: BOOL;
	mSuckertoRa AT %QX40.7: BOOL;
	//lightFurnance	--> NOT ASSIGNED
	compressor AT %QX41.0: BOOL;
	valveVacuum AT %QX41.1: BOOL;
	valveLowering AT %QX41.2: BOOL;
	valveFurnanceDoor AT %QX41.3: BOOL;
	valveSlider AT %QX41.4: BOOL;
	
	//------------------------------------------------------------------------------------//
	//------------------------------------PROGRAM VARS------------------------------------//
	//------------------------------------------------------------------------------------//
	// true if any motor/compressor of FUR is running
	any_motor_running: BOOL;
	
	// the state in which FUR currently is
	state: FUR_State;
	
	// BatchJob index in BatchJobQueue
	bIdxBurner: INT;
	bIdxSuccer: INT;
	bIdxSaw: INT;
	
	// workpiece index in current BatchJob
	wIdxBurner: INT;
	wIdxSuccer: INT;
	wIdxSaw: INT;
	
	// current workpieces
	currWBurner: Workpiece;
	currWSuccer: Workpiece;
	currWSaw: Workpiece;
END_VAR

// Device/Application/SL/SL
VAR_GLOBAL
	//------------------------------------------------------------------------------------//
	//--------------------------------------INPUTS----------------------------------------//
	//------------------------------------------------------------------------------------//
	iFeeler				AT %IX301.1: BOOL;
	lbEntry				AT %IX301.2: BOOL;
	lbAfterColorSensor	AT %IX301.3: BOOL;
	colorSensor 		AT %ID37: DINT; //analog
	lbWhite				AT %IX301.5: BOOL;
	lbRed				AT %IX301.6: BOOL;
	lbBlue				AT %IX301.7: BOOL;
	
	//------------------------------------------------------------------------------------//
	//--------------------------------------OUTPUTS---------------------------------------//
	//------------------------------------------------------------------------------------//	
	mConveyorBelt		AT %QX41.5: BOOL;
	compressor			AT %QX41.6: BOOL;
	valveFirstEject		AT %QX41.7: BOOL;
	valveSecEject		AT %QX41.7: BOOL;
	valveThirdEject		AT %QX41.7: BOOL;
	
	//------------------------------------------------------------------------------------//
	//------------------------------------PROGRAM VARS------------------------------------//
	//------------------------------------------------------------------------------------//
	// true if any motor or compressor of SL is running
	any_motor_running: BOOL;
	
	// the state in which SL currently is
	state: SL_State;
	
	// current BatchJob and workpiece index being processed at SL
	bIdx: INT;
	wIdx: INT;
	currW: Workpiece;
END_VAR

// Device/Application/VG/VG
VAR_GLOBAL
	//------------------------------------------------------------------------------------//
	//--------------------------------------INPUTS----------------------------------------//
	//------------------------------------------------------------------------------------//
	// s = switch
	sVertical AT %IX0.6: BOOL;
	sHorizontal AT %IX0.7: BOOL;
	sRotation AT %IX1.0: BOOL;
	// enc = encoder
	encVertical AT %IX1.3: BOOL;
	encHorizontal AT %IX1.4: BOOL;
	encRotation AT %IX1.5: BOOL;
	
	//------------------------------------------------------------------------------------//
	//--------------------------------------OUTPUTS---------------------------------------//
	//------------------------------------------------------------------------------------//	
	// m = motor
	mVerticalUp AT %QX1.0: BOOL;
	mVerticalDown AT %QX1.1: BOOL;
	mHorizontalBackward AT %QX1.2: BOOL;
	mHorizontalForward AT %QX1.3: BOOL;
	mRotationClockwise AT %QX1.4: BOOL;
	mRotationCClockwise AT %QX1.5: BOOL;
	compressor AT %QX1.6: BOOL;
	valve AT %QX1.7: BOOL;
	
	//------------------------------------------------------------------------------------//
	//------------------------------------PROGRAM VARS------------------------------------//
	//------------------------------------------------------------------------------------//
	// the state in which VG currently is
	state: VG_State;	
	
	// true if any motor of VG is running
	any_motor_running: BOOL;
	
	// flag used for decision making in multi mode
	storeW: BOOL;
	
	// counters defining the current position of VG
	cX: INT;
	cY: INT;
	cZ: INT;
	
	// current BatchJob and workpiece index being processed at VG
	bIdx: INT;
	wIdx: INT;
	currW: Workpiece;
END_VAR

// Device/Application/MAIN
PROGRAM MAIN
VAR_INPUT
END_VAR
VAR	
	workpieces: ARRAY [1..9] OF Workpiece;
	format: Format;
	format1: Format;
	format2: Format;
	format3: Format;
	format4: Format;
	format5: Format;
	format6: Format;
	format7: Format;
	format8: Format;
	format9: Format;
	format10: Format;
	format11: Format;
	format12: Format;
	format13: Format;
	format14: Format;
	format15: Format;
	format16: Format;
	newWorkpi: Workpiece;
END_VAR

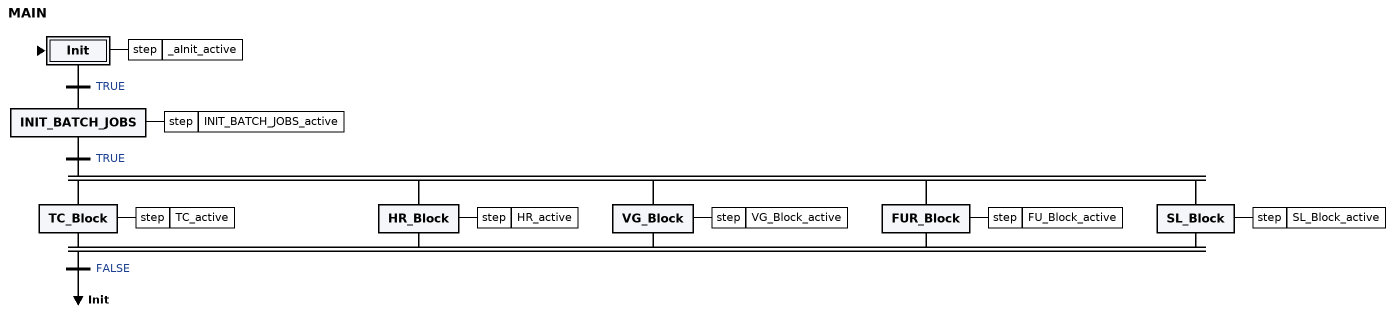
INITIAL_STEP Init:
    _aInit_active(N);  // step action
END_STEP
TRANSITION FROM Init TO INIT_BATCH_JOBS
    := TRUE;
END_TRANSITION
STEP INIT_BATCH_JOBS:
    INIT_BATCH_JOBS_active(N);  // step action
END_STEP
TRANSITION FROM INIT_BATCH_JOBS TO (TC_Block, HR_Block, VG_Block, FUR_Block, SL_Block)
    := TRUE;
END_TRANSITION
STEP TC_Block:
    TC_active(N);  // step action
END_STEP
STEP HR_Block:
    HR_active(N);  // step action
END_STEP
STEP VG_Block:
    VG_Block_active(N);  // step action
END_STEP
STEP FUR_Block:
    FU_Block_active(N);  // step action
END_STEP
STEP SL_Block:
    SL_Block_active(N);  // step action
END_STEP
TRANSITION FROM (TC_Block, HR_Block, VG_Block, FUR_Block, SL_Block) TO Init
    := FALSE;
END_TRANSITION

ACTION FU_Block_active:
(*
Copyright (c) 2019 Manuel Goester, Michael Witt, Klaus Kammerer
Institute of Databases and Information Systems, Ulm University, Germany

Permission is hereby granted, free of charge, to any person obtaining a copy 
of this software and associated documentation files (the "Software"), to deal 
in the Software without restriction, including without limitation the rights 
to use, copy, modify, merge, publish, distribute, sublicense, and/or sell 
copies of the Software, and to permit persons to whom the Software is 
furnished to do so, subject to the following conditions:

The above copyright notice and this permission notice shall be included in 
all copies or substantial portions of the Software.

THE SOFTWARE IS PROVIDED "AS IS", WITHOUT WARRANTY OF ANY KIND, EXPRESS OR 
IMPLIED, INCLUDING BUT NOT LIMITED TO THE WARRANTIES OF MERCHANTABILITY, 
FITNESS FOR A PARTICULAR PURPOSE AND NONINFRINGEMENT. IN NO EVENT SHALL THE 
AUTHORS OR COPYRIGHT HOLDERS BE LIABLE FOR ANY CLAIM, DAMAGES OR OTHER 
LIABILITY, WHETHER IN AN ACTION OF CONTRACT, TORT OR OTHERWISE, ARISING FROM, 
OUT OF OR IN CONNECTION WITH THE SOFTWARE OR THE USE OR OTHER DEALINGS 
IN THE SOFTWARE.
*)
FUR.any_motor_running := FUR.compressor AND FUR.mRaClockwise AND FUR.mRaCClockwise AND FUR.mConveyorBeltForward AND FUR.mSaw AND FUR.mFurnanceSliderIn  AND FUR.mFurnanceSliderOut AND FUR.mSuckertoFurnance AND FUR.mSuckertoRa AND FUR.compressor  AND FUR.valveVacuum AND FUR.valveLowering AND FUR.valveFurnanceDoor AND FUR.valveSlider;

IF (TC_POU.started OR FUR.any_motor_running) AND NOT(TC.instant_shutdown) THEN
	IF TC.mode_active = ExecutionMode.single THEN
		FUR_SINGLE_MODE();
	ELSIF TC.mode_active = ExecutionMode.multi THEN
		FUR_MULTI_MODE();
	END_IF
ELSE
	// instant shutdown --> all motors off
	FUR.compressor 				:= FALSE;
	FUR.mRaClockwise 			:= FALSE;
	FUR.mRaCClockwise  			:= FALSE;
	FUR.mConveyorBeltForward	:= FALSE;
	FUR.mSaw  					:= FALSE;
	FUR.mFurnanceSliderIn 		:= FALSE;
	FUR.mFurnanceSliderOut 		:= FALSE;
	FUR.mSuckertoFurnance 		:= FALSE;
	FUR.mSuckertoRa 			:= FALSE;
	FUR.compressor 				:= FALSE;
	FUR.valveVacuum				:= FALSE;
	FUR.valveLowering			:= FALSE;
	FUR.valveFurnanceDoor		:= FALSE;
	FUR.valveSlider 			:= FALSE;
END_IF
END_ACTION

ACTION VG_Block_active:
(*
Copyright (c) 2019 Manuel Goester, Michael Witt, Klaus Kammerer
Institute of Databases and Information Systems, Ulm University, Germany

Permission is hereby granted, free of charge, to any person obtaining a copy 
of this software and associated documentation files (the "Software"), to deal 
in the Software without restriction, including without limitation the rights 
to use, copy, modify, merge, publish, distribute, sublicense, and/or sell 
copies of the Software, and to permit persons to whom the Software is 
furnished to do so, subject to the following conditions:

The above copyright notice and this permission notice shall be included in 
all copies or substantial portions of the Software.

THE SOFTWARE IS PROVIDED "AS IS", WITHOUT WARRANTY OF ANY KIND, EXPRESS OR 
IMPLIED, INCLUDING BUT NOT LIMITED TO THE WARRANTIES OF MERCHANTABILITY, 
FITNESS FOR A PARTICULAR PURPOSE AND NONINFRINGEMENT. IN NO EVENT SHALL THE 
AUTHORS OR COPYRIGHT HOLDERS BE LIABLE FOR ANY CLAIM, DAMAGES OR OTHER 
LIABILITY, WHETHER IN AN ACTION OF CONTRACT, TORT OR OTHERWISE, ARISING FROM, 
OUT OF OR IN CONNECTION WITH THE SOFTWARE OR THE USE OR OTHER DEALINGS 
IN THE SOFTWARE.
*)
VG.any_motor_running := VG.mHorizontalBackward OR VG.mHorizontalForward OR VG.mRotationCClockwise OR VG.mRotationClockwise OR VG.mVerticalDown OR VG.mVerticalUp;

IF (TC_POU.started OR VG.any_motor_running) AND NOT(TC.instant_shutdown) THEN
	IF TC.mode_active = ExecutionMode.single THEN
		VG_SINGLE_MODE();
	ELSIF TC.mode_active = ExecutionMode.multi THEN
		VG_MULTI_MODE();
	END_IF
ELSE
	// instant shutdown --> all motors off
	VG.mHorizontalBackward 	:= FALSE;
	VG.mHorizontalForward 	:= FALSE;
	VG.mRotationCClockwise 	:= FALSE;
	VG.mRotationClockwise 	:= FALSE;
	VG.mVerticalDown 		:= FALSE; 
	VG.mVerticalUp 			:= FALSE;
END_IF
END_ACTION

ACTION SL_Block_active:
(*
Copyright (c) 2019 Manuel Goester, Michael Witt, Klaus Kammerer
Institute of Databases and Information Systems, Ulm University, Germany

Permission is hereby granted, free of charge, to any person obtaining a copy 
of this software and associated documentation files (the "Software"), to deal 
in the Software without restriction, including without limitation the rights 
to use, copy, modify, merge, publish, distribute, sublicense, and/or sell 
copies of the Software, and to permit persons to whom the Software is 
furnished to do so, subject to the following conditions:

The above copyright notice and this permission notice shall be included in 
all copies or substantial portions of the Software.

THE SOFTWARE IS PROVIDED "AS IS", WITHOUT WARRANTY OF ANY KIND, EXPRESS OR 
IMPLIED, INCLUDING BUT NOT LIMITED TO THE WARRANTIES OF MERCHANTABILITY, 
FITNESS FOR A PARTICULAR PURPOSE AND NONINFRINGEMENT. IN NO EVENT SHALL THE 
AUTHORS OR COPYRIGHT HOLDERS BE LIABLE FOR ANY CLAIM, DAMAGES OR OTHER 
LIABILITY, WHETHER IN AN ACTION OF CONTRACT, TORT OR OTHERWISE, ARISING FROM, 
OUT OF OR IN CONNECTION WITH THE SOFTWARE OR THE USE OR OTHER DEALINGS 
IN THE SOFTWARE.
*)
SL.any_motor_running := SL.mConveyorBelt AND SL.compressor;

IF (TC_POU.started OR SL.any_motor_running) AND NOT(TC.instant_shutdown) THEN
	IF TC.mode_active = ExecutionMode.single THEN
		SL_SINGLE_MODE();
	ELSIF TC.mode_active = ExecutionMode.multi THEN
		SL_MULTI_MODE();
	END_IF
ELSE
	// instant shutdown --> all motors off
	SL.mConveyorBelt 	:= FALSE;
	SL.compressor		:= FALSE;
END_IF
END_ACTION

ACTION TC_active:
(*
Copyright (c) 2019 Manuel Goester, Michael Witt, Klaus Kammerer
Institute of Databases and Information Systems, Ulm University, Germany

Permission is hereby granted, free of charge, to any person obtaining a copy 
of this software and associated documentation files (the "Software"), to deal 
in the Software without restriction, including without limitation the rights 
to use, copy, modify, merge, publish, distribute, sublicense, and/or sell 
copies of the Software, and to permit persons to whom the Software is 
furnished to do so, subject to the following conditions:

The above copyright notice and this permission notice shall be included in 
all copies or substantial portions of the Software.

THE SOFTWARE IS PROVIDED "AS IS", WITHOUT WARRANTY OF ANY KIND, EXPRESS OR 
IMPLIED, INCLUDING BUT NOT LIMITED TO THE WARRANTIES OF MERCHANTABILITY, 
FITNESS FOR A PARTICULAR PURPOSE AND NONINFRINGEMENT. IN NO EVENT SHALL THE 
AUTHORS OR COPYRIGHT HOLDERS BE LIABLE FOR ANY CLAIM, DAMAGES OR OTHER 
LIABILITY, WHETHER IN AN ACTION OF CONTRACT, TORT OR OTHERWISE, ARISING FROM, 
OUT OF OR IN CONNECTION WITH THE SOFTWARE OR THE USE OR OTHER DEALINGS 
IN THE SOFTWARE.
*)
// invoke TC_POU program
TC_POU();
END_ACTION

ACTION HR_active:
(*
Copyright (c) 2019 Manuel Goester, Michael Witt, Klaus Kammerer
Institute of Databases and Information Systems, Ulm University, Germany

Permission is hereby granted, free of charge, to any person obtaining a copy 
of this software and associated documentation files (the "Software"), to deal 
in the Software without restriction, including without limitation the rights 
to use, copy, modify, merge, publish, distribute, sublicense, and/or sell 
copies of the Software, and to permit persons to whom the Software is 
furnished to do so, subject to the following conditions:

The above copyright notice and this permission notice shall be included in 
all copies or substantial portions of the Software.

THE SOFTWARE IS PROVIDED "AS IS", WITHOUT WARRANTY OF ANY KIND, EXPRESS OR 
IMPLIED, INCLUDING BUT NOT LIMITED TO THE WARRANTIES OF MERCHANTABILITY, 
FITNESS FOR A PARTICULAR PURPOSE AND NONINFRINGEMENT. IN NO EVENT SHALL THE 
AUTHORS OR COPYRIGHT HOLDERS BE LIABLE FOR ANY CLAIM, DAMAGES OR OTHER 
LIABILITY, WHETHER IN AN ACTION OF CONTRACT, TORT OR OTHERWISE, ARISING FROM, 
OUT OF OR IN CONNECTION WITH THE SOFTWARE OR THE USE OR OTHER DEALINGS 
IN THE SOFTWARE.
*)
HR.any_motor_running := HR.mCBackward OR HR.mCForward OR HR.mCbBackward OR HR.mCbForward OR HR.mHorizontalLeft OR HR.mHorizontalRight OR HR.mVerticalDown OR HR.mVerticalUp;
// invoke the appropriate HR program that fits to the execution mode of the current batch job
IF (TC.batchJobQueue.batchJobs[TC.currBatchJobIdx].state = BatchJobState.STARTED OR HR.any_motor_running) AND NOT(TC.instant_shutdown) THEN
	IF TC.mode_active = ExecutionMode.single THEN
		HR_SINGLE_MODE();
	ELSIF TC.mode_active = ExecutionMode.multi THEN
		HR_MULTI_MODE();
	ELSIF TC.mode_active = ExecutionMode.sorting THEN
		HR.state := HR_State.SORTING;
		HR_SORTING_MODE();
	END_IF
ELSE
	// instant shutdown --> all motors off
	HR.mCBackward 		:= FALSE;
	HR.mCForward  		:= FALSE;
	HR.mCbBackward 		:= FALSE;
	HR.mCbForward  		:= FALSE;
	HR.mHorizontalLeft 	:= FALSE;
	HR.mHorizontalRight := FALSE;
	HR.mVerticalDown 	:= FALSE;
	HR.mVerticalUp 		:= FALSE;
END_IF
END_ACTION

ACTION _aInit_active:
(*
Copyright (c) 2019 Manuel Goester, Michael Witt, Klaus Kammerer
Institute of Databases and Information Systems, Ulm University, Germany

Permission is hereby granted, free of charge, to any person obtaining a copy 
of this software and associated documentation files (the "Software"), to deal 
in the Software without restriction, including without limitation the rights 
to use, copy, modify, merge, publish, distribute, sublicense, and/or sell 
copies of the Software, and to permit persons to whom the Software is 
furnished to do so, subject to the following conditions:

The above copyright notice and this permission notice shall be included in 
all copies or substantial portions of the Software.

THE SOFTWARE IS PROVIDED "AS IS", WITHOUT WARRANTY OF ANY KIND, EXPRESS OR 
IMPLIED, INCLUDING BUT NOT LIMITED TO THE WARRANTIES OF MERCHANTABILITY, 
FITNESS FOR A PARTICULAR PURPOSE AND NONINFRINGEMENT. IN NO EVENT SHALL THE 
AUTHORS OR COPYRIGHT HOLDERS BE LIABLE FOR ANY CLAIM, DAMAGES OR OTHER 
LIABILITY, WHETHER IN AN ACTION OF CONTRACT, TORT OR OTHERWISE, ARISING FROM, 
OUT OF OR IN CONNECTION WITH THE SOFTWARE OR THE USE OR OTHER DEALINGS 
IN THE SOFTWARE.
*)
// program has been started
TC.is_plc_running := TRUE;

// init some vars
TC.currBatchJobIdx := 1;
HR.any_motor_running := HR.mCBackward OR HR.mCForward OR HR.mCbBackward OR HR.mCbForward OR HR.mHorizontalLeft OR HR.mHorizontalRight OR HR.mVerticalDown OR HR.mVerticalUp;
VG.any_motor_running := VG.mHorizontalBackward OR VG.mHorizontalForward OR VG.mRotationCClockwise OR VG.mRotationClockwise OR VG.mVerticalDown OR VG.mVerticalUp;
FUR.any_motor_running := FUR.compressor AND FUR.mRaClockwise AND FUR.mRaCClockwise AND FUR.mConveyorBeltForward AND FUR.mSaw AND FUR.mFurnanceSliderIn  AND FUR.mFurnanceSliderOut AND FUR.mSuckertoFurnance AND FUR.mSuckertoRa AND FUR.compressor  AND FUR.valveVacuum AND FUR.valveLowering AND FUR.valveFurnanceDoor AND FUR.valveSlider;
SL.any_motor_running := SL.mConveyorBelt AND SL.compressor;
END_ACTION

ACTION INIT_BATCH_JOBS_active:
(*
	BatchJobs, which shall run on the DBIS Factory, will be initialized here
	By using the funciton TC_FUNs/addBatchJobToQueue a BatchJob can be added to the queue, e.g. by calling it via UA server

Copyright (c) 2019 Manuel Goester, Michael Witt, Klaus Kammerer
Institute of Databases and Information Systems, Ulm University, Germany

Permission is hereby granted, free of charge, to any person obtaining a copy 
of this software and associated documentation files (the "Software"), to deal 
in the Software without restriction, including without limitation the rights 
to use, copy, modify, merge, publish, distribute, sublicense, and/or sell 
copies of the Software, and to permit persons to whom the Software is 
furnished to do so, subject to the following conditions:

The above copyright notice and this permission notice shall be included in 
all copies or substantial portions of the Software.

THE SOFTWARE IS PROVIDED "AS IS", WITHOUT WARRANTY OF ANY KIND, EXPRESS OR 
IMPLIED, INCLUDING BUT NOT LIMITED TO THE WARRANTIES OF MERCHANTABILITY, 
FITNESS FOR A PARTICULAR PURPOSE AND NONINFRINGEMENT. IN NO EVENT SHALL THE 
AUTHORS OR COPYRIGHT HOLDERS BE LIABLE FOR ANY CLAIM, DAMAGES OR OTHER 
LIABILITY, WHETHER IN AN ACTION OF CONTRACT, TORT OR OTHERWISE, ARISING FROM, 
OUT OF OR IN CONNECTION WITH THE SOFTWARE OR THE USE OR OTHER DEALINGS 
IN THE SOFTWARE.
*)

(*
	Defining formats
*)
format1 := newFormat(FALSE, FALSE, FALSE, FALSE, T#5S, T#5S);
format2 := newFormat(FALSE, FALSE, FALSE, TRUE,  T#5S, T#5S);
format3 := newFormat(FALSE, FALSE, TRUE,  FALSE, T#5S, T#5S);
format4 := newFormat(FALSE, FALSE, TRUE,  TRUE,  T#5S, T#5S);

format5 := newFormat(FALSE, TRUE, FALSE, FALSE, T#5S, T#5S);
format6 := newFormat(FALSE, TRUE, FALSE, TRUE,  T#5S, T#5S);
format7 := newFormat(FALSE, TRUE, TRUE,  FALSE, T#5S, T#5S);
format8 := newFormat(FALSE, TRUE, TRUE,  TRUE,  T#5S, T#5S);

format9 := newFormat(TRUE, FALSE, FALSE, FALSE, T#5S, T#5S);
format10:= newFormat(TRUE, FALSE, FALSE, TRUE,  T#5S, T#5S);
format11:= newFormat(TRUE, FALSE, TRUE,  FALSE, T#5S, T#5S);
format12:= newFormat(TRUE, FALSE, TRUE,  TRUE,  T#5S, T#5S);

format13:= newFormat(TRUE, TRUE, FALSE, FALSE, T#5S, T#5S);
format14:= newFormat(TRUE, TRUE, FALSE, TRUE,  T#5S, T#5S);
format15:= newFormat(TRUE, TRUE, TRUE,  FALSE, T#5S, T#5S);
format16:= newFormat(TRUE, TRUE, TRUE,  TRUE,  T#5S, T#5S);

(*
	Testcase 1: SINGLE MODE
*)

workpieces[1] := newWorkpiece('unknown', W_State.AT_RACK_22, RackPos.RACK_22, RackPos.RACK_22, format15);
workpieces[2] := newWorkpiece('unknown', W_State.AT_RACK_23, RackPos.RACK_23, RackPos.RACK_23, format16);
workpieces[3] := newWorkpiece('unknown', W_State.AT_RACK_13, RackPos.RACK_13, RackPos.RACK_13, format8);
workpieces[4] := newWorkpiece('unknown', W_State.AT_RACK_21, RackPos.RACK_21, RackPos.RACK_21, format16);
workpieces[5] := newWorkpiece('unknown', W_State.AT_RACK_11, RackPos.RACK_11, RackPos.RACK_11, format15);
workpieces[6] := newWorkpiece('unknown', W_State.AT_RACK_12, RackPos.RACK_12, RackPos.RACK_12, format15);
addBatchJobToQueue(newbatchJob(6, workpieces, ExecutionMode.single));



(*
	Testcase 2: MULTI MODE
*)
(*
workpieces[1] := newWorkpiece('unknown', W_State.AT_RACK_22, RackPos.RACK_22, RackPos.RACK_22, format15);
workpieces[2] := newWorkpiece('unknown', W_State.AT_RACK_23, RackPos.RACK_23, RackPos.RACK_23, format16);
workpieces[3] := newWorkpiece('unknown', W_State.AT_RACK_13, RackPos.RACK_13, RackPos.RACK_13, format8);
workpieces[4] := newWorkpiece('unknown', W_State.AT_RACK_21, RackPos.RACK_21, RackPos.RACK_21, format16);
workpieces[5] := newWorkpiece('unknown', W_State.AT_RACK_11, RackPos.RACK_11, RackPos.RACK_11, format15);
workpieces[6] := newWorkpiece('unknown', W_State.AT_RACK_12, RackPos.RACK_12, RackPos.RACK_12, format15);
addBatchJobToQueue(newbatchJob(6, workpieces, ExecutionMode.multi));
*)


(*
	Testcase 3: SORTING MODE
*)
(*
workpieces[1] := newWorkpiece('unknown', W_State.AT_RACK_22, RackPos.RACK_22, RackPos.RACK_22, format15);
workpieces[2] := newWorkpiece('unknown', W_State.AT_RACK_23, RackPos.RACK_23, RackPos.RACK_23, format16);
workpieces[3] := newWorkpiece('unknown', W_State.AT_RACK_13, RackPos.RACK_13, RackPos.RACK_13, format8);
workpieces[4] := newWorkpiece('unknown', W_State.AT_RACK_21, RackPos.RACK_21, RackPos.RACK_21, format16);
addBatchJobToQueue(newbatchJob(4, workpieces, ExecutionMode.sorting));
*)
END_ACTION

END_PROGRAM

// Device/Application/TC/TC_POU
PROGRAM TC_POU
VAR
	// true if user pressed start button
	started: BOOL;
	
	// true if theres a batch job waiting to be executed
	batch_job_available: BOOL := FALSE;
	
	fin: BOOL;
	Copyright: INT;
END_VAR

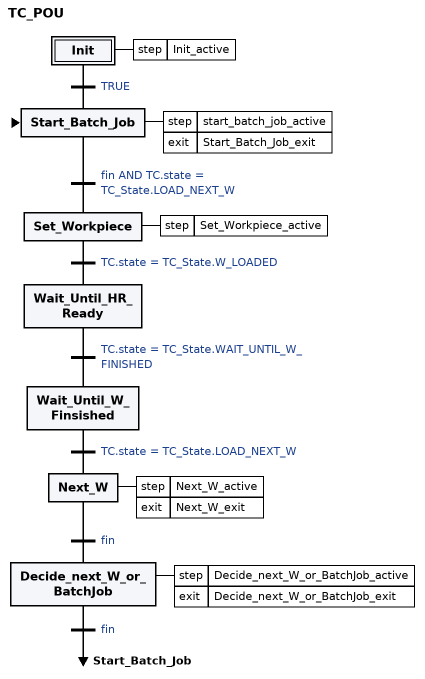
INITIAL_STEP Init:
    Init_active(N);  // step action
END_STEP
TRANSITION FROM Init TO Start_Batch_Job
    := TRUE;
END_TRANSITION
STEP Start_Batch_Job:
    start_batch_job_active(N);  // step action
    Start_Batch_Job_exit(P0);  // exit action
END_STEP
TRANSITION FROM Start_Batch_Job TO Set_Workpiece
    := fin AND TC.state = TC_State.LOAD_NEXT_W;
END_TRANSITION
STEP Set_Workpiece:
    Set_Workpiece_active(N);  // step action
END_STEP
TRANSITION FROM Set_Workpiece TO Wait_Until_HR_Ready
    := TC.state = TC_State.W_LOADED;
END_TRANSITION
STEP Wait_Until_HR_Ready:
END_STEP
TRANSITION FROM Wait_Until_HR_Ready TO Wait_Until_W_Finsished
    := TC.state = TC_State.WAIT_UNTIL_W_FINISHED;
END_TRANSITION
STEP Wait_Until_W_Finsished:
END_STEP
TRANSITION FROM Wait_Until_W_Finsished TO Next_W
    := TC.state = TC_State.LOAD_NEXT_W;
END_TRANSITION
STEP Next_W:
    	Next_W_active(N);  // step action
    Next_W_exit(P0);  // exit action
END_STEP
TRANSITION FROM Next_W TO Decide_next_W_or_BatchJob
    := fin;
END_TRANSITION
STEP Decide_next_W_or_BatchJob:
    Decide_next_W_or_BatchJob_active(N);  // step action
    Decide_next_W_or_BatchJob_exit(P0);  // exit action
END_STEP
TRANSITION FROM Decide_next_W_or_BatchJob TO Start_Batch_Job
    := fin;
END_TRANSITION

ACTION Decide_next_W_or_BatchJob_active:
(*
Copyright (c) 2019 Manuel Goester, Michael Witt, Klaus Kammerer
Institute of Databases and Information Systems, Ulm University, Germany

Permission is hereby granted, free of charge, to any person obtaining a copy 
of this software and associated documentation files (the "Software"), to deal 
in the Software without restriction, including without limitation the rights 
to use, copy, modify, merge, publish, distribute, sublicense, and/or sell 
copies of the Software, and to permit persons to whom the Software is 
furnished to do so, subject to the following conditions:

The above copyright notice and this permission notice shall be included in 
all copies or substantial portions of the Software.

THE SOFTWARE IS PROVIDED "AS IS", WITHOUT WARRANTY OF ANY KIND, EXPRESS OR 
IMPLIED, INCLUDING BUT NOT LIMITED TO THE WARRANTIES OF MERCHANTABILITY, 
FITNESS FOR A PARTICULAR PURPOSE AND NONINFRINGEMENT. IN NO EVENT SHALL THE 
AUTHORS OR COPYRIGHT HOLDERS BE LIABLE FOR ANY CLAIM, DAMAGES OR OTHER 
LIABILITY, WHETHER IN AN ACTION OF CONTRACT, TORT OR OTHERWISE, ARISING FROM, 
OUT OF OR IN CONNECTION WITH THE SOFTWARE OR THE USE OR OTHER DEALINGS 
IN THE SOFTWARE.
*)
IF NOT(fin) THEN
	IF TC.batchJobQueue.batchJobs[TC.currBatchJobIdx].nextNotProcessedIdx > TC.batchJobQueue.batchJobs[TC.currBatchJobIdx].batchSize THEN
		IF SM.currW.state = 0 AND HR.bIdx = 0 AND VG.bIdx = 0 AND FUR.bIdxBurner = 0 AND FUR.bIdxSuccer = 0 AND FUR.bIdxSaw = 0 AND SL.bIdx = 0 THEN
			// there is no new workpiece in current BatchJob and all maschines finished processing --> BatchJob finished
			TC.batchJobQueue.batchJobs[TC.currBatchJobIdx].state := BatchJobState.FINISHED;
			// delete finished BatchJob
			TC.batchJobQueue.batchJobs[TC.currBatchJobIdx] := TC.nullB;
			// update counter of BatchJobs in queue
			TC.batchJobQueue.amountBatchJobs := TC.batchJobQueue.amountBatchJobs - 1;
			// start next batch job if there is one
			TC.currBatchJobIdx := TC.currBatchJobIdx + 1;
			IF TC.currBatchJobIdx > 20 THEN
				TC.currBatchJobIdx := 1;
			END_IF
			fin := TRUE;
		END_IF
	ELSE
		// batch job not finished --> execute steps for next workpiece
		fin := TRUE;
	END_IF
END_IF
END_ACTION

ACTION Set_Workpiece_active:
(*
Copyright (c) 2019 Manuel Goester, Michael Witt, Klaus Kammerer
Institute of Databases and Information Systems, Ulm University, Germany

Permission is hereby granted, free of charge, to any person obtaining a copy 
of this software and associated documentation files (the "Software"), to deal 
in the Software without restriction, including without limitation the rights 
to use, copy, modify, merge, publish, distribute, sublicense, and/or sell 
copies of the Software, and to permit persons to whom the Software is 
furnished to do so, subject to the following conditions:

The above copyright notice and this permission notice shall be included in 
all copies or substantial portions of the Software.

THE SOFTWARE IS PROVIDED "AS IS", WITHOUT WARRANTY OF ANY KIND, EXPRESS OR 
IMPLIED, INCLUDING BUT NOT LIMITED TO THE WARRANTIES OF MERCHANTABILITY, 
FITNESS FOR A PARTICULAR PURPOSE AND NONINFRINGEMENT. IN NO EVENT SHALL THE 
AUTHORS OR COPYRIGHT HOLDERS BE LIABLE FOR ANY CLAIM, DAMAGES OR OTHER 
LIABILITY, WHETHER IN AN ACTION OF CONTRACT, TORT OR OTHERWISE, ARISING FROM, 
OUT OF OR IN CONNECTION WITH THE SOFTWARE OR THE USE OR OTHER DEALINGS 
IN THE SOFTWARE.
*)
IF TC.batchJobQueue.batchJobs[TC.currBatchJobIdx].state = BatchJobState.NULL THEN
	// no batchjob available
	// wait until new batchjob is loaded
ELSIF TC.batchJobQueue.batchJobs[TC.currBatchJobIdx].mode = ExecutionMode.single THEN
	SM.currW := TC.batchJobQueue.batchJobs[TC.currBatchJobIdx].workpieces[TC.batchJobQueue.batchJobs[TC.currBatchJobIdx].nextNotProcessedIdx];
	IF SM.currW.format.ejectEnabled AND NOT(SM.currW.format.furEnabled) AND NOT(SM.currW.format.sawEnabled) AND NOT(SM.currW.format.colorCheckEnabled) THEN
		// dont set SL flags because workpiece will directly be ejected HR -> VG -> EJECT
		SL.bIdx := 0;
		SL.wIdx := 0;
	ELSE
		// set SL pointers
		SL.bIdx := TC.currBatchJobIdx;
		SL.wIdx := TC.batchJobQueue.batchJobs[TC.currBatchJobIdx].nextNotProcessedIdx;
	END_IF
	TC.state := TC_State.W_LOADED;
ELSIF TC.batchJobQueue.batchJobs[TC.currBatchJobIdx].mode = ExecutionMode.multi AND (HR.state = HR_State.READY OR HR.state = HR_State.FINISHED_SINGLE_MODE OR HR.state = HR_State.SORTING) THEN
	// new w loaded in TC, load it to HR.currW
	Hr.bIdx := TC.currBatchJobIdx;
	Hr.wIdx := TC.batchJobQueue.batchJobs[TC.currBatchJobIdx].nextNotProcessedIdx;
	HR.currW := TC.batchJobQueue.batchJobs[Hr.bIdx].workpieces[Hr.wIdx];
	TC.state := TC_State.W_LOADED;
ELSIF TC.batchJobQueue.batchJobs[TC.currBatchJobIdx].mode = ExecutionMode.sorting THEN
	TC.state := TC_State.W_LOADED;
END_IF
END_ACTION

ACTION start_batch_job_active:
(*
Copyright (c) 2019 Manuel Goester, Michael Witt, Klaus Kammerer
Institute of Databases and Information Systems, Ulm University, Germany

Permission is hereby granted, free of charge, to any person obtaining a copy 
of this software and associated documentation files (the "Software"), to deal 
in the Software without restriction, including without limitation the rights 
to use, copy, modify, merge, publish, distribute, sublicense, and/or sell 
copies of the Software, and to permit persons to whom the Software is 
furnished to do so, subject to the following conditions:

The above copyright notice and this permission notice shall be included in 
all copies or substantial portions of the Software.

THE SOFTWARE IS PROVIDED "AS IS", WITHOUT WARRANTY OF ANY KIND, EXPRESS OR 
IMPLIED, INCLUDING BUT NOT LIMITED TO THE WARRANTIES OF MERCHANTABILITY, 
FITNESS FOR A PARTICULAR PURPOSE AND NONINFRINGEMENT. IN NO EVENT SHALL THE 
AUTHORS OR COPYRIGHT HOLDERS BE LIABLE FOR ANY CLAIM, DAMAGES OR OTHER 
LIABILITY, WHETHER IN AN ACTION OF CONTRACT, TORT OR OTHERWISE, ARISING FROM, 
OUT OF OR IN CONNECTION WITH THE SOFTWARE OR THE USE OR OTHER DEALINGS 
IN THE SOFTWARE.
*)
IF started THEN
	IF NOT(fin) THEN
		IF TC.batchJobQueue.batchJobs[TC.currBatchJobIdx].state <> BatchJobState.NULL THEN
			IF TC.batchJobQueue.batchJobs[TC.currBatchJobIdx].mode = ExecutionMode.single THEN
				// start single mode
				TC.mode_active := ExecutionMode.single;
				TC.batchJobQueue.batchJobs[TC.currBatchJobIdx].state := BatchJobState.STARTED;
				fin := TRUE;
			ELSIF TC.batchJobQueue.batchJobs[TC.currBatchJobIdx].mode = ExecutionMode.multi THEN
				// start multi mode
				TC.mode_active := ExecutionMode.multi;
				TC.batchJobQueue.batchJobs[TC.currBatchJobIdx].state := BatchJobState.STARTED;
				fin := TRUE;
			ELSIF TC.batchJobQueue.batchJobs[TC.currBatchJobIdx].mode = ExecutionMode.sorting THEN
				// start sorting mode
				TC.mode_active := ExecutionMode.sorting;
				TC.batchJobQueue.batchJobs[TC.currBatchJobIdx].state := BatchJobState.STARTED;
				fin := TRUE;
			END_IF
		ELSE
			// currently no BatchJob available
			// reset HR pointers, cause they may still set
			HR.bIdx := 0;
			HR.wIdx := 0;
			HR.currW := TC.nullW;
		END_IF
	END_IF
END_IF
END_ACTION

ACTION Init_active:
(*
Copyright (c) 2019 Manuel Goester, Michael Witt, Klaus Kammerer
Institute of Databases and Information Systems, Ulm University, Germany

Permission is hereby granted, free of charge, to any person obtaining a copy 
of this software and associated documentation files (the "Software"), to deal 
in the Software without restriction, including without limitation the rights 
to use, copy, modify, merge, publish, distribute, sublicense, and/or sell 
copies of the Software, and to permit persons to whom the Software is 
furnished to do so, subject to the following conditions:

The above copyright notice and this permission notice shall be included in 
all copies or substantial portions of the Software.

THE SOFTWARE IS PROVIDED "AS IS", WITHOUT WARRANTY OF ANY KIND, EXPRESS OR 
IMPLIED, INCLUDING BUT NOT LIMITED TO THE WARRANTIES OF MERCHANTABILITY, 
FITNESS FOR A PARTICULAR PURPOSE AND NONINFRINGEMENT. IN NO EVENT SHALL THE 
AUTHORS OR COPYRIGHT HOLDERS BE LIABLE FOR ANY CLAIM, DAMAGES OR OTHER 
LIABILITY, WHETHER IN AN ACTION OF CONTRACT, TORT OR OTHERWISE, ARISING FROM, 
OUT OF OR IN CONNECTION WITH THE SOFTWARE OR THE USE OR OTHER DEALINGS 
IN THE SOFTWARE.
*)
TC.state := TC_State.NULL;
END_ACTION

ACTION Next_W_active:
(*
Copyright (c) 2019 Manuel Goester, Michael Witt, Klaus Kammerer
Institute of Databases and Information Systems, Ulm University, Germany

Permission is hereby granted, free of charge, to any person obtaining a copy 
of this software and associated documentation files (the "Software"), to deal 
in the Software without restriction, including without limitation the rights 
to use, copy, modify, merge, publish, distribute, sublicense, and/or sell 
copies of the Software, and to permit persons to whom the Software is 
furnished to do so, subject to the following conditions:

The above copyright notice and this permission notice shall be included in 
all copies or substantial portions of the Software.

THE SOFTWARE IS PROVIDED "AS IS", WITHOUT WARRANTY OF ANY KIND, EXPRESS OR 
IMPLIED, INCLUDING BUT NOT LIMITED TO THE WARRANTIES OF MERCHANTABILITY, 
FITNESS FOR A PARTICULAR PURPOSE AND NONINFRINGEMENT. IN NO EVENT SHALL THE 
AUTHORS OR COPYRIGHT HOLDERS BE LIABLE FOR ANY CLAIM, DAMAGES OR OTHER 
LIABILITY, WHETHER IN AN ACTION OF CONTRACT, TORT OR OTHERWISE, ARISING FROM, 
OUT OF OR IN CONNECTION WITH THE SOFTWARE OR THE USE OR OTHER DEALINGS 
IN THE SOFTWARE.
*)
// updates the current workpiece pointer to the next workpiece
IF NOT(fin) THEN
	IF NOT(TC.batchJobQueue.batchJobs[TC.currBatchJobIdx].mode = ExecutionMode.sorting) THEN
		TC.batchJobQueue.batchJobs[TC.currBatchJobIdx].nextNotProcessedIdx := TC.batchJobQueue.batchJobs[TC.currBatchJobIdx].nextNotProcessedIdx + 1;
	ELSE
		// in sorting mode always two workpieces are processed simultaniously, so increment by 2
		TC.batchJobQueue.batchJobs[TC.currBatchJobIdx].nextNotProcessedIdx := TC.batchJobQueue.batchJobs[TC.currBatchJobIdx].nextNotProcessedIdx + 2;
	END_IF
	fin := TRUE;
END_IF
END_ACTION

ACTION Next_W_exit:
(*
Copyright (c) 2019 Manuel Goester, Michael Witt, Klaus Kammerer
Institute of Databases and Information Systems, Ulm University, Germany

Permission is hereby granted, free of charge, to any person obtaining a copy 
of this software and associated documentation files (the "Software"), to deal 
in the Software without restriction, including without limitation the rights 
to use, copy, modify, merge, publish, distribute, sublicense, and/or sell 
copies of the Software, and to permit persons to whom the Software is 
furnished to do so, subject to the following conditions:

The above copyright notice and this permission notice shall be included in 
all copies or substantial portions of the Software.

THE SOFTWARE IS PROVIDED "AS IS", WITHOUT WARRANTY OF ANY KIND, EXPRESS OR 
IMPLIED, INCLUDING BUT NOT LIMITED TO THE WARRANTIES OF MERCHANTABILITY, 
FITNESS FOR A PARTICULAR PURPOSE AND NONINFRINGEMENT. IN NO EVENT SHALL THE 
AUTHORS OR COPYRIGHT HOLDERS BE LIABLE FOR ANY CLAIM, DAMAGES OR OTHER 
LIABILITY, WHETHER IN AN ACTION OF CONTRACT, TORT OR OTHERWISE, ARISING FROM, 
OUT OF OR IN CONNECTION WITH THE SOFTWARE OR THE USE OR OTHER DEALINGS 
IN THE SOFTWARE.
*)
fin := FALSE;
END_ACTION

ACTION Decide_next_W_or_BatchJob_exit:
(*
Copyright (c) 2019 Manuel Goester, Michael Witt, Klaus Kammerer
Institute of Databases and Information Systems, Ulm University, Germany

Permission is hereby granted, free of charge, to any person obtaining a copy 
of this software and associated documentation files (the "Software"), to deal 
in the Software without restriction, including without limitation the rights 
to use, copy, modify, merge, publish, distribute, sublicense, and/or sell 
copies of the Software, and to permit persons to whom the Software is 
furnished to do so, subject to the following conditions:

The above copyright notice and this permission notice shall be included in 
all copies or substantial portions of the Software.

THE SOFTWARE IS PROVIDED "AS IS", WITHOUT WARRANTY OF ANY KIND, EXPRESS OR 
IMPLIED, INCLUDING BUT NOT LIMITED TO THE WARRANTIES OF MERCHANTABILITY, 
FITNESS FOR A PARTICULAR PURPOSE AND NONINFRINGEMENT. IN NO EVENT SHALL THE 
AUTHORS OR COPYRIGHT HOLDERS BE LIABLE FOR ANY CLAIM, DAMAGES OR OTHER 
LIABILITY, WHETHER IN AN ACTION OF CONTRACT, TORT OR OTHERWISE, ARISING FROM, 
OUT OF OR IN CONNECTION WITH THE SOFTWARE OR THE USE OR OTHER DEALINGS 
IN THE SOFTWARE.
*)
fin := FALSE;
END_ACTION

ACTION Start_Batch_Job_exit:
(*
Copyright (c) 2019 Manuel Goester, Michael Witt, Klaus Kammerer
Institute of Databases and Information Systems, Ulm University, Germany

Permission is hereby granted, free of charge, to any person obtaining a copy 
of this software and associated documentation files (the "Software"), to deal 
in the Software without restriction, including without limitation the rights 
to use, copy, modify, merge, publish, distribute, sublicense, and/or sell 
copies of the Software, and to permit persons to whom the Software is 
furnished to do so, subject to the following conditions:

The above copyright notice and this permission notice shall be included in 
all copies or substantial portions of the Software.

THE SOFTWARE IS PROVIDED "AS IS", WITHOUT WARRANTY OF ANY KIND, EXPRESS OR 
IMPLIED, INCLUDING BUT NOT LIMITED TO THE WARRANTIES OF MERCHANTABILITY, 
FITNESS FOR A PARTICULAR PURPOSE AND NONINFRINGEMENT. IN NO EVENT SHALL THE 
AUTHORS OR COPYRIGHT HOLDERS BE LIABLE FOR ANY CLAIM, DAMAGES OR OTHER 
LIABILITY, WHETHER IN AN ACTION OF CONTRACT, TORT OR OTHERWISE, ARISING FROM, 
OUT OF OR IN CONNECTION WITH THE SOFTWARE OR THE USE OR OTHER DEALINGS 
IN THE SOFTWARE.
*)
fin := FALSE;
END_ACTION

END_PROGRAM

// Device/Application/FUR/FUR_SINGLE_MODE
PROGRAM FUR_SINGLE_MODE
VAR
	trigger: INT;
	timer: TON;
	sawStopped: BOOL;
	wAtSL: BOOL;
	fin: BOOL;
END_VAR

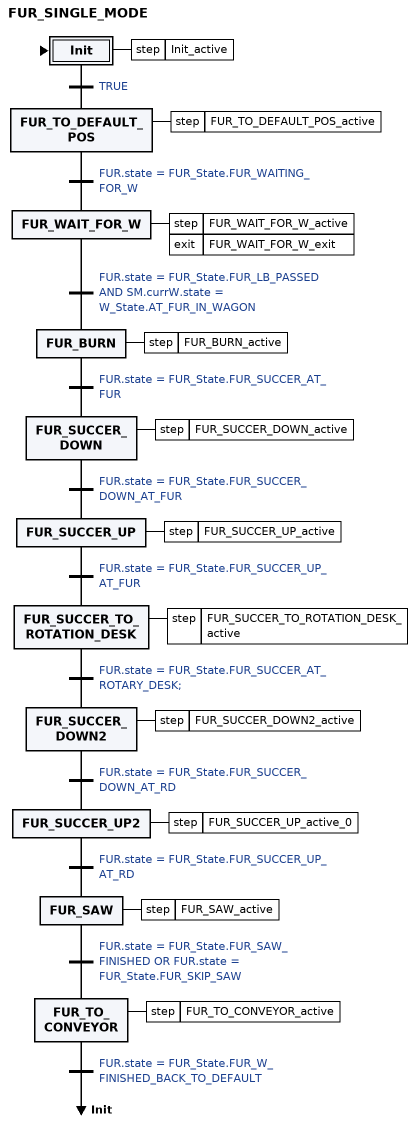
INITIAL_STEP Init:
    Init_active(N);  // step action
END_STEP
TRANSITION FROM Init TO FUR_TO_DEFAULT_POS
    := TRUE;
END_TRANSITION
STEP FUR_TO_DEFAULT_POS:
    FUR_TO_DEFAULT_POS_active(N);  // step action
END_STEP
TRANSITION FROM FUR_TO_DEFAULT_POS TO FUR_WAIT_FOR_W
    := FUR.state = FUR_State.FUR_WAITING_FOR_W;
END_TRANSITION
STEP FUR_WAIT_FOR_W:
    FUR_WAIT_FOR_W_active(N);  // step action
    FUR_WAIT_FOR_W_exit(P0);  // exit action
END_STEP
TRANSITION FROM FUR_WAIT_FOR_W TO FUR_BURN
    := FUR.state = FUR_State.FUR_LB_PASSED AND SM.currW.state = W_State.AT_FUR_IN_WAGON;
END_TRANSITION
STEP FUR_BURN:
    FUR_BURN_active(N);  // step action
END_STEP
TRANSITION FROM FUR_BURN TO FUR_SUCCER_DOWN
    := FUR.state = FUR_State.FUR_SUCCER_AT_FUR;
END_TRANSITION
STEP FUR_SUCCER_DOWN:
    FUR_SUCCER_DOWN_active(N);  // step action
END_STEP
TRANSITION FROM FUR_SUCCER_DOWN TO FUR_SUCCER_UP
    := FUR.state = FUR_State.FUR_SUCCER_DOWN_AT_FUR;
END_TRANSITION
STEP FUR_SUCCER_UP:
    FUR_SUCCER_UP_active(N);  // step action
END_STEP
TRANSITION FROM FUR_SUCCER_UP TO FUR_SUCCER_TO_ROTATION_DESK
    := FUR.state = FUR_State.FUR_SUCCER_UP_AT_FUR;
END_TRANSITION
STEP FUR_SUCCER_TO_ROTATION_DESK:
    FUR_SUCCER_TO_ROTATION_DESK_active(N);  // step action
END_STEP
TRANSITION FROM FUR_SUCCER_TO_ROTATION_DESK TO FUR_SUCCER_DOWN2
    := FUR.state = FUR_State.FUR_SUCCER_AT_ROTARY_DESK;
END_TRANSITION
STEP FUR_SUCCER_DOWN2:
    FUR_SUCCER_DOWN2_active(N);  // step action
END_STEP
TRANSITION FROM FUR_SUCCER_DOWN2 TO FUR_SUCCER_UP2
    := FUR.state = FUR_State.FUR_SUCCER_DOWN_AT_RD;
END_TRANSITION
STEP FUR_SUCCER_UP2:
    FUR_SUCCER_UP_active_0(N);  // step action
END_STEP
TRANSITION FROM FUR_SUCCER_UP2 TO FUR_SAW
    := FUR.state = FUR_State.FUR_SUCCER_UP_AT_RD;
END_TRANSITION
STEP FUR_SAW:
    FUR_SAW_active(N);  // step action
END_STEP
TRANSITION FROM FUR_SAW TO FUR_TO_CONVEYOR
    := FUR.state = FUR_State.FUR_SAW_FINISHED OR FUR.state = FUR_State.FUR_SKIP_SAW;
END_TRANSITION
STEP FUR_TO_CONVEYOR:
    FUR_TO_CONVEYOR_active(N);  // step action
END_STEP
TRANSITION FROM FUR_TO_CONVEYOR TO Init
    := FUR.state = FUR_State.FUR_W_FINISHED_BACK_TO_DEFAULT;
END_TRANSITION

ACTION FUR_SUCCER_UP_active_0:
(*
Copyright (c) 2019 Manuel Goester, Michael Witt, Klaus Kammerer
Institute of Databases and Information Systems, Ulm University, Germany

Permission is hereby granted, free of charge, to any person obtaining a copy 
of this software and associated documentation files (the "Software"), to deal 
in the Software without restriction, including without limitation the rights 
to use, copy, modify, merge, publish, distribute, sublicense, and/or sell 
copies of the Software, and to permit persons to whom the Software is 
furnished to do so, subject to the following conditions:

The above copyright notice and this permission notice shall be included in 
all copies or substantial portions of the Software.

THE SOFTWARE IS PROVIDED "AS IS", WITHOUT WARRANTY OF ANY KIND, EXPRESS OR 
IMPLIED, INCLUDING BUT NOT LIMITED TO THE WARRANTIES OF MERCHANTABILITY, 
FITNESS FOR A PARTICULAR PURPOSE AND NONINFRINGEMENT. IN NO EVENT SHALL THE 
AUTHORS OR COPYRIGHT HOLDERS BE LIABLE FOR ANY CLAIM, DAMAGES OR OTHER 
LIABILITY, WHETHER IN AN ACTION OF CONTRACT, TORT OR OTHERWISE, ARISING FROM, 
OUT OF OR IN CONNECTION WITH THE SOFTWARE OR THE USE OR OTHER DEALINGS 
IN THE SOFTWARE.
*)
timer(IN:= TRUE, PT := T#200MS);
IF NOT(timer.Q = FALSE AND timer.IN) THEN
	timer(IN:= FALSE);
	FUR.state := FUR_State.FUR_SUCCER_UP_AT_RD;
	SM.currW.state := W_State.AT_FUR_ON_ROTARY_DESK;
END_IF
END_ACTION

ACTION FUR_SUCCER_TO_ROTATION_DESK_active:
(*
Copyright (c) 2019 Manuel Goester, Michael Witt, Klaus Kammerer
Institute of Databases and Information Systems, Ulm University, Germany

Permission is hereby granted, free of charge, to any person obtaining a copy 
of this software and associated documentation files (the "Software"), to deal 
in the Software without restriction, including without limitation the rights 
to use, copy, modify, merge, publish, distribute, sublicense, and/or sell 
copies of the Software, and to permit persons to whom the Software is 
furnished to do so, subject to the following conditions:

The above copyright notice and this permission notice shall be included in 
all copies or substantial portions of the Software.

THE SOFTWARE IS PROVIDED "AS IS", WITHOUT WARRANTY OF ANY KIND, EXPRESS OR 
IMPLIED, INCLUDING BUT NOT LIMITED TO THE WARRANTIES OF MERCHANTABILITY, 
FITNESS FOR A PARTICULAR PURPOSE AND NONINFRINGEMENT. IN NO EVENT SHALL THE 
AUTHORS OR COPYRIGHT HOLDERS BE LIABLE FOR ANY CLAIM, DAMAGES OR OTHER 
LIABILITY, WHETHER IN AN ACTION OF CONTRACT, TORT OR OTHERWISE, ARISING FROM, 
OUT OF OR IN CONNECTION WITH THE SOFTWARE OR THE USE OR OTHER DEALINGS 
IN THE SOFTWARE.
*)
IF  NOT(FUR.sSuckerPosRa) THEN
	FUR.mSuckertoRa := TRUE;
	FUR.state := FUR_State.FUR_SUCCER_TO_ROTARY_DESK;
ELSE
	FUR.mSuckertoRa := FALSE;
	FUR.compressor := FALSE;
	FUR.valveLowering := TRUE;
	FUR.state := FUR_State.FUR_SUCCER_AT_ROTARY_DESK;
END_IF
END_ACTION

ACTION FUR_SAW_active:
(*
Copyright (c) 2019 Manuel Goester, Michael Witt, Klaus Kammerer
Institute of Databases and Information Systems, Ulm University, Germany

Permission is hereby granted, free of charge, to any person obtaining a copy 
of this software and associated documentation files (the "Software"), to deal 
in the Software without restriction, including without limitation the rights 
to use, copy, modify, merge, publish, distribute, sublicense, and/or sell 
copies of the Software, and to permit persons to whom the Software is 
furnished to do so, subject to the following conditions:

The above copyright notice and this permission notice shall be included in 
all copies or substantial portions of the Software.

THE SOFTWARE IS PROVIDED "AS IS", WITHOUT WARRANTY OF ANY KIND, EXPRESS OR 
IMPLIED, INCLUDING BUT NOT LIMITED TO THE WARRANTIES OF MERCHANTABILITY, 
FITNESS FOR A PARTICULAR PURPOSE AND NONINFRINGEMENT. IN NO EVENT SHALL THE 
AUTHORS OR COPYRIGHT HOLDERS BE LIABLE FOR ANY CLAIM, DAMAGES OR OTHER 
LIABILITY, WHETHER IN AN ACTION OF CONTRACT, TORT OR OTHERWISE, ARISING FROM, 
OUT OF OR IN CONNECTION WITH THE SOFTWARE OR THE USE OR OTHER DEALINGS 
IN THE SOFTWARE.
*)
IF SM.currW.format.sawEnabled THEN
	SM.currW.state := W_State.AT_FUR_AT_SAW;
	IF NOT(FUR.sRaPosSaw) THEN
		FUR.mRaClockwise := TRUE;
	ELSE
		FUR.mRaClockwise := FALSE;
		sawStopped := TRUE;
	END_IF
	
	IF sawStopped THEN
		timer(IN:= TRUE, PT := SM.currW.format.sawDuration);
		FUR.mSaw := TRUE;
		
		IF NOT(timer.Q = FALSE AND timer.IN) THEN
			timer(IN:=FALSE);
			FUR.mSaw := FALSE;
			sawStopped := FALSE;
			FUR.state := FUR_State.FUR_SAW_FINISHED;
		END_IF
	END_IF
ELSE
	// skip saw
	FUR.state := FUR_State.FUR_SKIP_SAW;
END_IF
END_ACTION

ACTION FUR_WAIT_FOR_W_exit:
(*
Copyright (c) 2019 Manuel Goester, Michael Witt, Klaus Kammerer
Institute of Databases and Information Systems, Ulm University, Germany

Permission is hereby granted, free of charge, to any person obtaining a copy 
of this software and associated documentation files (the "Software"), to deal 
in the Software without restriction, including without limitation the rights 
to use, copy, modify, merge, publish, distribute, sublicense, and/or sell 
copies of the Software, and to permit persons to whom the Software is 
furnished to do so, subject to the following conditions:

The above copyright notice and this permission notice shall be included in 
all copies or substantial portions of the Software.

THE SOFTWARE IS PROVIDED "AS IS", WITHOUT WARRANTY OF ANY KIND, EXPRESS OR 
IMPLIED, INCLUDING BUT NOT LIMITED TO THE WARRANTIES OF MERCHANTABILITY, 
FITNESS FOR A PARTICULAR PURPOSE AND NONINFRINGEMENT. IN NO EVENT SHALL THE 
AUTHORS OR COPYRIGHT HOLDERS BE LIABLE FOR ANY CLAIM, DAMAGES OR OTHER 
LIABILITY, WHETHER IN AN ACTION OF CONTRACT, TORT OR OTHERWISE, ARISING FROM, 
OUT OF OR IN CONNECTION WITH THE SOFTWARE OR THE USE OR OTHER DEALINGS 
IN THE SOFTWARE.
*)
trigger := 0;
END_ACTION

ACTION Init_active:
(*
Copyright (c) 2019 Manuel Goester, Michael Witt, Klaus Kammerer
Institute of Databases and Information Systems, Ulm University, Germany

Permission is hereby granted, free of charge, to any person obtaining a copy 
of this software and associated documentation files (the "Software"), to deal 
in the Software without restriction, including without limitation the rights 
to use, copy, modify, merge, publish, distribute, sublicense, and/or sell 
copies of the Software, and to permit persons to whom the Software is 
furnished to do so, subject to the following conditions:

The above copyright notice and this permission notice shall be included in 
all copies or substantial portions of the Software.

THE SOFTWARE IS PROVIDED "AS IS", WITHOUT WARRANTY OF ANY KIND, EXPRESS OR 
IMPLIED, INCLUDING BUT NOT LIMITED TO THE WARRANTIES OF MERCHANTABILITY, 
FITNESS FOR A PARTICULAR PURPOSE AND NONINFRINGEMENT. IN NO EVENT SHALL THE 
AUTHORS OR COPYRIGHT HOLDERS BE LIABLE FOR ANY CLAIM, DAMAGES OR OTHER 
LIABILITY, WHETHER IN AN ACTION OF CONTRACT, TORT OR OTHERWISE, ARISING FROM, 
OUT OF OR IN CONNECTION WITH THE SOFTWARE OR THE USE OR OTHER DEALINGS 
IN THE SOFTWARE.
*)
FUR.state := -1;
sawStopped := FALSE;
trigger := 0;
END_ACTION

ACTION FUR_SUCCER_DOWN2_active:
(*
Copyright (c) 2019 Manuel Goester, Michael Witt, Klaus Kammerer
Institute of Databases and Information Systems, Ulm University, Germany

Permission is hereby granted, free of charge, to any person obtaining a copy 
of this software and associated documentation files (the "Software"), to deal 
in the Software without restriction, including without limitation the rights 
to use, copy, modify, merge, publish, distribute, sublicense, and/or sell 
copies of the Software, and to permit persons to whom the Software is 
furnished to do so, subject to the following conditions:

The above copyright notice and this permission notice shall be included in 
all copies or substantial portions of the Software.

THE SOFTWARE IS PROVIDED "AS IS", WITHOUT WARRANTY OF ANY KIND, EXPRESS OR 
IMPLIED, INCLUDING BUT NOT LIMITED TO THE WARRANTIES OF MERCHANTABILITY, 
FITNESS FOR A PARTICULAR PURPOSE AND NONINFRINGEMENT. IN NO EVENT SHALL THE 
AUTHORS OR COPYRIGHT HOLDERS BE LIABLE FOR ANY CLAIM, DAMAGES OR OTHER 
LIABILITY, WHETHER IN AN ACTION OF CONTRACT, TORT OR OTHERWISE, ARISING FROM, 
OUT OF OR IN CONNECTION WITH THE SOFTWARE OR THE USE OR OTHER DEALINGS 
IN THE SOFTWARE.
*)
IF FUR.sFurnanceSliderOutside THEN
	FUR.compressor := TRUE;
	FUR.valveLowering := TRUE;
	FUR.valveVacuum := FALSE;
	timer(IN:= TRUE, PT := T#1S);
	IF NOT(timer.Q = FALSE AND timer.IN) THEN
		timer(IN:= FALSE);
		FUR.valveLowering := FALSE;
		FUR.state := FUR_State.FUR_SUCCER_DOWN_AT_RD;
	END_IF
END_IF
END_ACTION

ACTION FUR_SUCCER_DOWN_active:
(*
Copyright (c) 2019 Manuel Goester, Michael Witt, Klaus Kammerer
Institute of Databases and Information Systems, Ulm University, Germany

Permission is hereby granted, free of charge, to any person obtaining a copy 
of this software and associated documentation files (the "Software"), to deal 
in the Software without restriction, including without limitation the rights 
to use, copy, modify, merge, publish, distribute, sublicense, and/or sell 
copies of the Software, and to permit persons to whom the Software is 
furnished to do so, subject to the following conditions:

The above copyright notice and this permission notice shall be included in 
all copies or substantial portions of the Software.

THE SOFTWARE IS PROVIDED "AS IS", WITHOUT WARRANTY OF ANY KIND, EXPRESS OR 
IMPLIED, INCLUDING BUT NOT LIMITED TO THE WARRANTIES OF MERCHANTABILITY, 
FITNESS FOR A PARTICULAR PURPOSE AND NONINFRINGEMENT. IN NO EVENT SHALL THE 
AUTHORS OR COPYRIGHT HOLDERS BE LIABLE FOR ANY CLAIM, DAMAGES OR OTHER 
LIABILITY, WHETHER IN AN ACTION OF CONTRACT, TORT OR OTHERWISE, ARISING FROM, 
OUT OF OR IN CONNECTION WITH THE SOFTWARE OR THE USE OR OTHER DEALINGS 
IN THE SOFTWARE.
*)
timer(IN:= TRUE, PT := T#2S);
//sauger zum ofen
IF FUR.sFurnanceSliderOutside THEN
	FUR.compressor := TRUE;
	FUR.valveLowering := TRUE;
END_IF

IF NOT(timer.Q = FALSE AND timer.IN) THEN
	// reset timer
	timer(IN:= FALSE);
	// go to next step
	FUR.state := FUR_State.FUR_SUCCER_DOWN_AT_FUR;
END_IF
END_ACTION

ACTION FUR_TO_CONVEYOR_active:
(*
Copyright (c) 2019 Manuel Goester, Michael Witt, Klaus Kammerer
Institute of Databases and Information Systems, Ulm University, Germany

Permission is hereby granted, free of charge, to any person obtaining a copy 
of this software and associated documentation files (the "Software"), to deal 
in the Software without restriction, including without limitation the rights 
to use, copy, modify, merge, publish, distribute, sublicense, and/or sell 
copies of the Software, and to permit persons to whom the Software is 
furnished to do so, subject to the following conditions:

The above copyright notice and this permission notice shall be included in 
all copies or substantial portions of the Software.

THE SOFTWARE IS PROVIDED "AS IS", WITHOUT WARRANTY OF ANY KIND, EXPRESS OR 
IMPLIED, INCLUDING BUT NOT LIMITED TO THE WARRANTIES OF MERCHANTABILITY, 
FITNESS FOR A PARTICULAR PURPOSE AND NONINFRINGEMENT. IN NO EVENT SHALL THE 
AUTHORS OR COPYRIGHT HOLDERS BE LIABLE FOR ANY CLAIM, DAMAGES OR OTHER 
LIABILITY, WHETHER IN AN ACTION OF CONTRACT, TORT OR OTHERWISE, ARISING FROM, 
OUT OF OR IN CONNECTION WITH THE SOFTWARE OR THE USE OR OTHER DEALINGS 
IN THE SOFTWARE.
*)
SM.currW.state := W_State.AT_FUR_ON_CONVEYOR;
SL.state := SL_State.W_RECEIVED;
IF NOT(FUR.sRaPosConveyorBelt) THEN
	FUR.mRaClockwise := TRUE;
ELSE
	FUR.mRaClockwise := FALSE;
	FUR.compressor := TRUE;
	FUR.valveSlider := TRUE;
END_IF

IF SL.lbEntry THEN
	FUR.mConveyorBeltForward := TRUE;
ELSE
	FUR.mConveyorBeltForward := FALSE;
	FUR.compressor := FALSE;
	FUR.valveSlider := FALSE;
	FUR.state := FUR_State.FUR_W_FINISHED_BACK_TO_DEFAULT;
END_IF
END_ACTION

ACTION FUR_SUCCER_UP_active:
(*
Copyright (c) 2019 Manuel Goester, Michael Witt, Klaus Kammerer
Institute of Databases and Information Systems, Ulm University, Germany

Permission is hereby granted, free of charge, to any person obtaining a copy 
of this software and associated documentation files (the "Software"), to deal 
in the Software without restriction, including without limitation the rights 
to use, copy, modify, merge, publish, distribute, sublicense, and/or sell 
copies of the Software, and to permit persons to whom the Software is 
furnished to do so, subject to the following conditions:

The above copyright notice and this permission notice shall be included in 
all copies or substantial portions of the Software.

THE SOFTWARE IS PROVIDED "AS IS", WITHOUT WARRANTY OF ANY KIND, EXPRESS OR 
IMPLIED, INCLUDING BUT NOT LIMITED TO THE WARRANTIES OF MERCHANTABILITY, 
FITNESS FOR A PARTICULAR PURPOSE AND NONINFRINGEMENT. IN NO EVENT SHALL THE 
AUTHORS OR COPYRIGHT HOLDERS BE LIABLE FOR ANY CLAIM, DAMAGES OR OTHER 
LIABILITY, WHETHER IN AN ACTION OF CONTRACT, TORT OR OTHERWISE, ARISING FROM, 
OUT OF OR IN CONNECTION WITH THE SOFTWARE OR THE USE OR OTHER DEALINGS 
IN THE SOFTWARE.
*)
FUR.valveLowering := FALSE;
FUR.valveVacuum := TRUE; //hier, sonst wird kein vakuum erzeugt
SM.currW.state := W_State.AT_FUR_ATTACHED_TO_SUCCER;
FUR.state := FUR_State.FUR_SUCCER_UP_AT_FUR;
END_ACTION

ACTION FUR_TO_DEFAULT_POS_active:
(*
Copyright (c) 2019 Manuel Goester, Michael Witt, Klaus Kammerer
Institute of Databases and Information Systems, Ulm University, Germany

Permission is hereby granted, free of charge, to any person obtaining a copy 
of this software and associated documentation files (the "Software"), to deal 
in the Software without restriction, including without limitation the rights 
to use, copy, modify, merge, publish, distribute, sublicense, and/or sell 
copies of the Software, and to permit persons to whom the Software is 
furnished to do so, subject to the following conditions:

The above copyright notice and this permission notice shall be included in 
all copies or substantial portions of the Software.

THE SOFTWARE IS PROVIDED "AS IS", WITHOUT WARRANTY OF ANY KIND, EXPRESS OR 
IMPLIED, INCLUDING BUT NOT LIMITED TO THE WARRANTIES OF MERCHANTABILITY, 
FITNESS FOR A PARTICULAR PURPOSE AND NONINFRINGEMENT. IN NO EVENT SHALL THE 
AUTHORS OR COPYRIGHT HOLDERS BE LIABLE FOR ANY CLAIM, DAMAGES OR OTHER 
LIABILITY, WHETHER IN AN ACTION OF CONTRACT, TORT OR OTHERWISE, ARISING FROM, 
OUT OF OR IN CONNECTION WITH THE SOFTWARE OR THE USE OR OTHER DEALINGS 
IN THE SOFTWARE.
*)
IF NOT(FUR.sFurnanceSliderOutside) THEN
	FUR.mFurnanceSliderOut := TRUE;
ELSE
	FUR.mFurnanceSliderOut := FALSE;
END_IF

IF NOT(FUR.sSuckerPosRa) THEN
	FUR.mSuckertoRa := TRUE;
ELSE
	FUR.mSuckertoRa := FALSE;
END_IF

IF NOT(FUR.sRaPosSucker) THEN
	FUR.mRaCClockwise := TRUE;
ELSE
	FUR.mRaCClockwise := FALSE;
END_IF

IF FUR.sSuckerPosRa AND FUR.sRaPosSucker AND FUR.sFurnanceSliderOutside THEN
	FUR.state := FUR_WAITING_FOR_W;
END_IF
END_ACTION

ACTION FUR_WAIT_FOR_W_active:
(*
Copyright (c) 2019 Manuel Goester, Michael Witt, Klaus Kammerer
Institute of Databases and Information Systems, Ulm University, Germany

Permission is hereby granted, free of charge, to any person obtaining a copy 
of this software and associated documentation files (the "Software"), to deal 
in the Software without restriction, including without limitation the rights 
to use, copy, modify, merge, publish, distribute, sublicense, and/or sell 
copies of the Software, and to permit persons to whom the Software is 
furnished to do so, subject to the following conditions:

The above copyright notice and this permission notice shall be included in 
all copies or substantial portions of the Software.

THE SOFTWARE IS PROVIDED "AS IS", WITHOUT WARRANTY OF ANY KIND, EXPRESS OR 
IMPLIED, INCLUDING BUT NOT LIMITED TO THE WARRANTIES OF MERCHANTABILITY, 
FITNESS FOR A PARTICULAR PURPOSE AND NONINFRINGEMENT. IN NO EVENT SHALL THE 
AUTHORS OR COPYRIGHT HOLDERS BE LIABLE FOR ANY CLAIM, DAMAGES OR OTHER 
LIABILITY, WHETHER IN AN ACTION OF CONTRACT, TORT OR OTHERWISE, ARISING FROM, 
OUT OF OR IN CONNECTION WITH THE SOFTWARE OR THE USE OR OTHER DEALINGS 
IN THE SOFTWARE.
*)
// Workpiece passes the light barrier
IF NOT(FUR.lbFurnance) AND trigger < 2 THEN
	trigger := trigger + 1;
END_IF

// Workpiece passed light barrier
IF FUR.lbFurnance AND trigger >= 2 THEN
	FUR.state := FUR_State.FUR_LB_PASSED;
END_IF
END_ACTION

ACTION FUR_BURN_active:
(*
Copyright (c) 2019 Manuel Goester, Michael Witt, Klaus Kammerer
Institute of Databases and Information Systems, Ulm University, Germany

Permission is hereby granted, free of charge, to any person obtaining a copy 
of this software and associated documentation files (the "Software"), to deal 
in the Software without restriction, including without limitation the rights 
to use, copy, modify, merge, publish, distribute, sublicense, and/or sell 
copies of the Software, and to permit persons to whom the Software is 
furnished to do so, subject to the following conditions:

The above copyright notice and this permission notice shall be included in 
all copies or substantial portions of the Software.

THE SOFTWARE IS PROVIDED "AS IS", WITHOUT WARRANTY OF ANY KIND, EXPRESS OR 
IMPLIED, INCLUDING BUT NOT LIMITED TO THE WARRANTIES OF MERCHANTABILITY, 
FITNESS FOR A PARTICULAR PURPOSE AND NONINFRINGEMENT. IN NO EVENT SHALL THE 
AUTHORS OR COPYRIGHT HOLDERS BE LIABLE FOR ANY CLAIM, DAMAGES OR OTHER 
LIABILITY, WHETHER IN AN ACTION OF CONTRACT, TORT OR OTHERWISE, ARISING FROM, 
OUT OF OR IN CONNECTION WITH THE SOFTWARE OR THE USE OR OTHER DEALINGS 
IN THE SOFTWARE.
*)
IF SM.currW.format.furEnabled THEN
	// open door and drive workpiece into furnance 
	IF FUR.state = FUR_State.FUR_LB_PASSED THEN
		FUR.compressor := TRUE;
		FUR.valveFurnanceDoor := TRUE;
		IF FUR.sFurnanceSliderInside = FALSE THEN
			FUR.mFurnanceSliderIn := TRUE;
		ELSE
			FUR.mFurnanceSliderIn := FALSE;
			FUR.state := FUR_State.FUR_WAGON_INSIDE;
		END_IF
	END_IF
	
	// burn
	IF FUR.state = FUR_State.FUR_WAGON_INSIDE THEN
		SM.currW.state := W_State.AT_FUR_IN_FUR;
		timer(IN:= TRUE, PT := SM.currW.format.furDuration);
		FUR.valveFurnanceDoor := FALSE;
		trigger := 0;
		
		// timer finished
		IF NOT(timer.Q = FALSE AND timer.IN) THEN
			timer(IN:= FALSE);
			FUR.compressor := TRUE;
			FUR.valveFurnanceDoor := TRUE;
			FUR.state := FUR_State.FUR_BURNED;
		END_IF
	END_IF
	
	// drive slider out
	IF FUR.state = FUR_State.FUR_BURNED THEN
		SM.currW.state := W_State.AT_FUR_IN_WAGON;
		IF FUR.sFurnanceSliderOutside = FALSE THEN
			FUR.mFurnanceSliderOut := TRUE;
		ELSE
			FUR.mFurnanceSliderOut := FALSE;
			FUR.state := FUR_State.FUR_WAGON_OUTSIDE;
		END_IF
	END_IF
	
	
	// bring succer to furnace
	IF NOT(FUR.sSuckerPosFF) AND (FUR.state = FUR_State.FUR_WAGON_INSIDE OR FUR.state = FUR_State.FUR_BURNED OR FUR.state = FUR_State.FUR_WAGON_OUTSIDE) THEN
		FUR.mSuckertoFurnance := TRUE;
	ELSE
		FUR.mSuckertoFurnance := FALSE;
	END_IF
	
	IF FUR.state = FUR_State.FUR_WAGON_OUTSIDE AND FUR.sSuckerPosFF THEN
		FUR.state := FUR_State.FUR_SUCCER_AT_FUR;
		FUR.mFurnanceSliderOut := FALSE;
		FUR.compressor := FALSE;
		FUR.valveFurnanceDoor := FALSE;
	END_IF
	
ELSE	
	// skip burning
	// bring succer to furnance
	IF NOT(FUR.sSuckerPosFF) THEN
		FUR.mSuckertoFurnance := TRUE;
	ELSE
		FUR.mSuckertoFurnance := FALSE;
		FUR.state := FUR_State.FUR_SUCCER_AT_FUR;
	END_IF
END_IF
END_ACTION

END_PROGRAM

// Device/Application/FUR/FUR_MULTI_MODE
PROGRAM FUR_MULTI_MODE
VAR
	fur_burn: FUR_BURN;
	timer: TON;
	finBurner: BOOL := FALSE;
	stepSuccer: INT := 1;
	stepSaw: INT := 1;
	fin: BOOL;
	counter: INT;
END_VAR

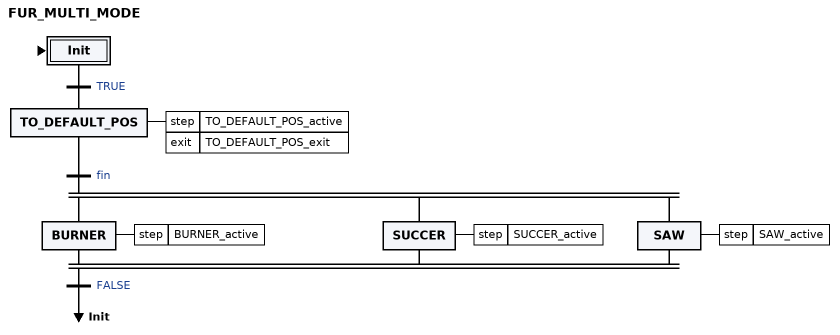
INITIAL_STEP Init:
END_STEP
TRANSITION FROM Init TO TO_DEFAULT_POS
    := TRUE;
END_TRANSITION
STEP TO_DEFAULT_POS:
    TO_DEFAULT_POS_active(N);  // step action
    TO_DEFAULT_POS_exit(P0);  // exit action
END_STEP
TRANSITION FROM TO_DEFAULT_POS TO (BURNER, SUCCER, SAW)
    := fin;
END_TRANSITION
STEP BURNER:
    BURNER_active(N);  // step action
END_STEP
STEP SUCCER:
    SUCCER_active(N);  // step action
END_STEP
STEP SAW:
    SAW_active(N);  // step action
END_STEP
TRANSITION FROM (BURNER, SUCCER, SAW) TO Init
    := FALSE;
END_TRANSITION

ACTION BURNER_active:
(*
Copyright (c) 2019 Manuel Goester, Michael Witt, Klaus Kammerer
Institute of Databases and Information Systems, Ulm University, Germany

Permission is hereby granted, free of charge, to any person obtaining a copy 
of this software and associated documentation files (the "Software"), to deal 
in the Software without restriction, including without limitation the rights 
to use, copy, modify, merge, publish, distribute, sublicense, and/or sell 
copies of the Software, and to permit persons to whom the Software is 
furnished to do so, subject to the following conditions:

The above copyright notice and this permission notice shall be included in 
all copies or substantial portions of the Software.

THE SOFTWARE IS PROVIDED "AS IS", WITHOUT WARRANTY OF ANY KIND, EXPRESS OR 
IMPLIED, INCLUDING BUT NOT LIMITED TO THE WARRANTIES OF MERCHANTABILITY, 
FITNESS FOR A PARTICULAR PURPOSE AND NONINFRINGEMENT. IN NO EVENT SHALL THE 
AUTHORS OR COPYRIGHT HOLDERS BE LIABLE FOR ANY CLAIM, DAMAGES OR OTHER 
LIABILITY, WHETHER IN AN ACTION OF CONTRACT, TORT OR OTHERWISE, ARISING FROM, 
OUT OF OR IN CONNECTION WITH THE SOFTWARE OR THE USE OR OTHER DEALINGS 
IN THE SOFTWARE.
*)
IF FUR.currWBurner.state <> W_State.NULL THEN
	// fur burner got an w
	IF FUR.currWBurner.format.furEnabled AND NOT(finBurner) THEN
		// burn
		fur_burn(w := FUR.currWBurner);
		finBurner := fur_burn.fin;
	ELSE
		IF FUR.currWSuccer.state = W_State.NULL THEN
			// bend pointers of fur succer to current workpiece
			counter := counter + 1;
			
			FUR.bIdxSuccer := FUR.bIdxBurner;
			FUR.wIdxSuccer := FUR.wIdxBurner;
			FUR.currWSuccer := TC.batchJobQueue.batchJobs[FUR.bIdxSuccer].workpieces[FUR.wIdxSuccer];
			// reset own pointers
			FUR.bIdxBurner := 0;
			FUR.wIdxBurner := 0;
			FUR.currWBurner := TC.nullW;
			finBurner := FALSE;
		END_IF
	END_IF
END_IF
END_ACTION

ACTION SUCCER_active:
(*
Copyright (c) 2019 Manuel Goester, Michael Witt, Klaus Kammerer
Institute of Databases and Information Systems, Ulm University, Germany

Permission is hereby granted, free of charge, to any person obtaining a copy 
of this software and associated documentation files (the "Software"), to deal 
in the Software without restriction, including without limitation the rights 
to use, copy, modify, merge, publish, distribute, sublicense, and/or sell 
copies of the Software, and to permit persons to whom the Software is 
furnished to do so, subject to the following conditions:

The above copyright notice and this permission notice shall be included in 
all copies or substantial portions of the Software.

THE SOFTWARE IS PROVIDED "AS IS", WITHOUT WARRANTY OF ANY KIND, EXPRESS OR 
IMPLIED, INCLUDING BUT NOT LIMITED TO THE WARRANTIES OF MERCHANTABILITY, 
FITNESS FOR A PARTICULAR PURPOSE AND NONINFRINGEMENT. IN NO EVENT SHALL THE 
AUTHORS OR COPYRIGHT HOLDERS BE LIABLE FOR ANY CLAIM, DAMAGES OR OTHER 
LIABILITY, WHETHER IN AN ACTION OF CONTRACT, TORT OR OTHERWISE, ARISING FROM, 
OUT OF OR IN CONNECTION WITH THE SOFTWARE OR THE USE OR OTHER DEALINGS 
IN THE SOFTWARE.
*)
CASE stepSuccer OF
	1:	
		IF FUR.currWBurner.state <> W_State.NULL OR FUR.currWSuccer.state <> W_State.NULL THEN
			stepSuccer := stepSuccer + 1;
		ELSE
			// do nothing, because w will not be sawed or color checked, so VG will bring w back to HR or to EJECT after burning
		END_IF
	2:
		// fur succer got an w --> pick it up and bring it to saw
		// bring succer to furnace
		IF NOT(FUR.sSuckerPosFF) THEN
			FUR.mSuckertoFurnance := TRUE;
		ELSE
			FUR.mSuckertoFurnance := FALSE;
			stepSuccer := stepSuccer + 1;
		END_IF
	3:
		// succer at waggon and rotation desk at succer pos, bring succer down to pick up w
		IF FUR.sFurnanceSliderOutside AND FUR.sRaPosSucker THEN
			FUR.compressor := TRUE;
			FUR.valveLowering := TRUE;
			timer(IN:= TRUE, PT := T#2S);
			IF NOT(timer.Q = FALSE AND timer.IN) THEN
				// reset timer
				timer(IN:= FALSE);
				// go to next step
				//FUR.state := FUR_State.FUR_SUCCER_DOWN_AT_FUR;
				stepSuccer := stepSuccer + 1;
			END_IF
		END_IF
	4: 
		// succer at waggon, succed w, pick up w
		FUR.valveLowering := FALSE;
		FUR.valveVacuum := TRUE; // otherwise vacuum will not be created
		//SM.currW.state := StateEnum.AT_FUR_ATTACHED_TO_SUCCER;
		//FUR.state := FUR_State.FUR_SUCCER_UP_AT_FUR;
		stepSuccer := stepSuccer + 1;
	5:
		// succer to rotation desk
		IF  NOT(FUR.sSuckerPosRa) THEN
			FUR.mSuckertoRa := TRUE;
			//FUR.state := FUR_State.FUR_SUCCER_TO_ROTARY_DESK;
		ELSE
			FUR.mSuckertoRa := FALSE;
			FUR.compressor := FALSE;
			FUR.valveLowering := TRUE;
			//FUR.state := FUR_State.FUR_SUCCER_AT_ROTARY_DESK;
			stepSuccer := stepSuccer + 1;
		END_IF
	6:
		// succer at rotation desk, bring succer down in order to put down w
		IF FUR.sFurnanceSliderOutside THEN
			FUR.compressor := TRUE;
			FUR.valveLowering := TRUE;
			FUR.valveVacuum := FALSE;
			timer(IN:= TRUE, PT := T#1S);
			IF NOT(timer.Q = FALSE AND timer.IN) THEN
				timer(IN:= FALSE);
				FUR.valveLowering := FALSE;
				//FUR.state := FUR_State.FUR_SUCCER_DOWN_AT_RD;
				stepSuccer := stepSuccer + 1;
			END_IF
		END_IF
	7:
		// wait 200ms before rotating desk
		timer(IN:= TRUE, PT := T#200MS);
		IF NOT(timer.Q = FALSE AND timer.IN) THEN
			timer(IN:= FALSE);
			//FUR.state := FUR_State.FUR_SUCCER_UP_AT_RD;
			//SM.currW.state := W_State.AT_FUR_ON_ROTARY_DESK;
			stepSuccer := stepSuccer + 1;
		END_IF
	8:
		IF FUR.currWSaw.state = W_State.NULL THEN
			// bend pointers of saw to current workpiece
			FUR.bIdxSaw := FUR.bIdxSuccer;
			FUR.wIdxSaw := FUR.wIdxSuccer;
			FUR.currWSaw := TC.batchJobQueue.batchJobs[FUR.bIdxSaw].workpieces[FUR.wIdxSaw];
			// reset own pointers
			FUR.bIdxSuccer := 0;
			FUR.wIdxSuccer := 0;
			FUR.currWSuccer := TC.nullW;
			// finsihed, go back to 1 to wait for next w
			stepSuccer := 1;
		ELSE
			// wait for saw to be ready to take a new w
		END_IF
		
END_CASE
END_ACTION

